LIN {X 0,Y 270.682,Z 565.079,A -85,B 0,C 180,E1 -18602.136,E2 -18602.136} C_VEL
LIN {X 0,Y 267.95,Z 577.412,A -85,B 0,C 180,E1 -18603.937,E2 -18603.937} C_VEL
LIN {X 0,Y 265.369,Z 587.551,A -85,B 0,C 180,E1 -18605.762,E2 -18605.762} C_VEL
LIN {X 0,Y 262.729,Z 597.619,A -85,B 0,C 180,E1 -18608.005,E2 -18608.005} C_VEL
LIN {X 0,Y 260.354,Z 605.98,A -85,B 0,C 180,E1 -18610.278,E2 -18610.278} C_VEL
LIN {X 0,Y 258.26,Z 613.967,A -85,B 0,C 180,E1 -18612.988,E2 -18612.988} C_VEL
LIN {X 0,Y 257.055,Z 618.72,A -85,B 0,C 180,E1 -18614.944,E2 -18614.944} C_VEL
LIN {X 0,Y 255.748,Z 623.456,A -85,B 0,C 180,E1 -18617.298,E2 -18617.298} C_VEL
LIN {X 0,Y 254.729,Z 628.359,A -85,B 0,C 180,E1 -18620.469,E2 -18620.469} C_VEL
LIN {X 0,Y 254.16,Z 631.774,A -85,B 0,C 180,E1 -18623.648,E2 -18623.648} C_VEL
LIN {X 0,Y 253.922,Z 633.804,A -85,B 0,C 180,E1 -18626.825,E2 -18626.825} C_VEL
LIN {X 0,Y 253.945,Z 634.498,A -85,B 0,C 180,E1 -18629.998,E2 -18629.998} C_VEL
LIN {X 0,Y 253.921,Z 633.866,A -85,B 0,C 180,E1 -18633.171,E2 -18633.171} C_VEL
LIN {X 0,Y 254.158,Z 631.893,A -85,B 0,C 180,E1 -18636.348,E2 -18636.348} C_VEL
LIN {X 0,Y 254.724,Z 628.531,A -85,B 0,C 180,E1 -18639.527,E2 -18639.527} C_VEL
LIN {X 0,Y 255.718,Z 623.68,A -85,B 0,C 180,E1 -18642.699,E2 -18642.699} C_VEL
LIN {X 0,Y 257.545,Z 617.197,A -85,B 0,C 180,E1 -18645.834,E2 -18645.834} C_VEL
LIN {X 0,Y 259.188,Z 610.543,A -85,B 0,C 180,E1 -18648.369,E2 -18648.369} C_VEL
LIN {X 0,Y 261.415,Z 602.415,A -85,B 0,C 180,E1 -18650.866,E2 -18650.866} C_VEL
LIN {X 0,Y 263.884,Z 593.336,A -85,B 0,C 180,E1 -18653.129,E2 -18653.129} C_VEL
LIN {X 0,Y 266.775,Z 582.336,A -85,B 0,C 180,E1 -18655.344,E2 -18655.344} C_VEL
LIN {X 0,Y 269.468,Z 571.253,A -85,B 0,C 180,E1 -18657.132,E2 -18657.132} C_VEL
LIN {X 0,Y 271.722,Z 560.272,A -85,B 0,C 180,E1 -18658.584,E2 -18658.584} C_VEL
LIN {X 0,Y 273.816,Z 548.655,A -85,B 0,C 180,E1 -18659.819,E2 -18659.819} C_VEL
LIN {X 0,Y 275.788,Z 536.139,A -85,B 0,C 180,E1 -18660.851,E2 -18660.851} C_VEL
LIN {X 0,Y 277.465,Z 522.233,A -85,B 0,C 180,E1 -18661.705,E2 -18661.705} C_VEL
LIN {X 0,Y 278.662,Z 508.127,A -85,B 0,C 180,E1 -18662.276,E2 -18662.276} C_VEL
LIN {X 0,Y 282.069,Z 423.35,A -85,B 0,C 180,E1 -18664.395,E2 -18664.395} C_VEL
LIN {X 0,Y 281.708,Z 421.592,A -85,B 0,C 180,E1 -18664.499,E2 -18664.499} C_VEL
LIN {X 0,Y 275.516,Z 406.79,A -85,B 0,C 180,E1 -18665.852,E2 -18665.852} C_VEL
LIN {X 0,Y 268.504,Z 392.298,A -85,B 0,C 180,E1 -18667.416,E2 -18667.416} C_VEL
LIN {X 0,Y 262.239,Z 380.582,A -85,B 0,C 180,E1 -18668.873,E2 -18668.873} C_VEL
LIN {X 0,Y 257.627,Z 372.309,A -85,B 0,C 180,E1 -18670.051,E2 -18670.051} C_VEL
LIN {X 0,Y 256.183,Z 367.432,A -85,B 0,C 180,E1 -18672.208,E2 -18672.208} C_VEL
LIN {X 0,Y 256.111,Z 367.17,A -85,B 0,C 180,E1 -18675.515,E2 -18675.515} C_VEL
LIN {X 0,Y 256.146,Z 367.192,A -85,B 0,C 180,E1 -18677.575,E2 -18677.575} C_VEL
LIN {X 0,Y 255.514,Z 367.285,A -85,B 0,C 180,E1 -18678.888,E2 -18678.888} C_VEL
LIN {X 0,Y 252.632,Z 367.623,A -85,B 0,C 180,E1 -18681.027,E2 -18681.027} C_VEL
LIN {X 0,Y 250.17,Z 367.909,A -85,B 0,C 180,E1 -18682.768,E2 -18682.768} C_VEL
LIN {X 0,Y 249.129,Z 368.043,A -85,B 0,C 180,E1 -18684.12,E2 -18684.12} C_VEL
LIN {X 0,Y 249.055,Z 368.06,A -85,B 0,C 180,E1 -18684.578,E2 -18684.578} C_VEL
LIN {X 0,Y 249.032,Z 368.067,A -85,B 0,C 180,E1 -18687.843,E2 -18687.843} C_VEL
LIN {X 0,Y 249.077,Z 368.015,A -85,B 0,C 180,E1 -18691.336,E2 -18691.336} C_VEL
LIN {X 0,Y 249.147,Z 368.069,A -85,B 0,C 180,E1 -18694.968,E2 -18694.968} C_VEL
LIN {X 0,Y 249.101,Z 368.069,A -85,B 0,C 180,E1 -18700.211,E2 -18700.211} C_VEL
LIN {X 0,Y 249.233,Z 368.043,A -85,B 0,C 180,E1 -18703.621,E2 -18703.621} C_VEL
LIN {X 0,Y 249.244,Z 368.052,A -85,B 0,C 180,E1 -18708.616,E2 -18708.616} C_VEL
LIN {X 0,Y 249.472,Z 368.017,A -85,B 0,C 180,E1 -18711.902,E2 -18711.902} C_VEL
LIN {X 0,Y 249.428,Z 368.015,A -85,B 0,C 180,E1 -18716.769,E2 -18716.769} C_VEL
LIN {X 0,Y 249.735,Z 368.002,A -85,B 0,C 180,E1 -18720,E2 -18720} C_VEL
LIN {X 0,Y 249.428,Z 368.015,A -85,B 0,C 180,E1 -18723.23,E2 -18723.23} C_VEL
LIN {X 0,Y 249.472,Z 368.018,A -85,B 0,C 180,E1 -18728.097,E2 -18728.097} C_VEL
LIN {X 0,Y 249.243,Z 368.05,A -85,B 0,C 180,E1 -18731.384,E2 -18731.384} C_VEL
LIN {X 0,Y 249.232,Z 368.041,A -85,B 0,C 180,E1 -18736.379,E2 -18736.379} C_VEL
LIN {X 0,Y 249.078,Z 368.062,A -85,B 0,C 180,E1 -18741.519,E2 -18741.519} C_VEL
LIN {X 0,Y 249.12,Z 368.062,A -85,B 0,C 180,E1 -18745.483,E2 -18745.483} C_VEL
LIN {X 0,Y 249.045,Z 368.017,A -85,B 0,C 180,E1 -18748.982,E2 -18748.982} C_VEL
LIN {X 0,Y 249.024,Z 368.074,A -85,B 0,C 180,E1 -18752.427,E2 -18752.427} C_VEL
LIN {X 0,Y 249.066,Z 368.042,A -85,B 0,C 180,E1 -18756.339,E2 -18756.339} C_VEL
LIN {X 0,Y 249.077,Z 368.064,A -85,B 0,C 180,E1 -18760.464,E2 -18760.464} C_VEL
LIN {X 0,Y 249.089,Z 368.062,A -85,B 0,C 180,E1 -18762.816,E2 -18762.816} C_VEL
LIN {X 0,Y 249.124,Z 368.184,A -85,B 0,C 180,E1 -18766.624,E2 -18766.624} C_VEL
LIN {X 0,Y 250.316,Z 372.193,A -85,B 0,C 180,E1 -18768.548,E2 -18768.548} C_VEL
LIN {X 0,Y 252.81,Z 376.584,A -85,B 0,C 180,E1 -18769.283,E2 -18769.283} C_VEL
LIN {X 0,Y 260.86,Z 390.951,A -85,B 0,C 180,E1 -18771.287,E2 -18771.287} C_VEL
LIN {X 0,Y 269.178,Z 407.825,A -85,B 0,C 180,E1 -18773.246,E2 -18773.246} C_VEL
LIN {X 0,Y 275.708,Z 423.186,A -85,B 0,C 180,E1 -18774.736,E2 -18774.736} C_VEL
LIN {X 0,Y 276.16,Z 424.395,A -85,B 0,C 180,E1 -18774.84,E2 -18774.84} C_VEL
LIN {X 0,Y 273.32,Z 494.281,A -85,B 0,C 180,E1 -18776.602,E2 -18776.602} C_VEL
LIN {X 0,Y 272.36,Z 512.78,A -85,B 0,C 180,E1 -18777.143,E2 -18777.143} C_VEL
LIN {X 0,Y 270.901,Z 526.969,A -85,B 0,C 180,E1 -18777.818,E2 -18777.818} C_VEL
LIN {X 0,Y 268.863,Z 541.315,A -85,B 0,C 180,E1 -18778.812,E2 -18778.812} C_VEL
LIN {X 0,Y 266.816,Z 553.585,A -85,B 0,C 180,E1 -18779.972,E2 -18779.972} C_VEL
LIN {X 0,Y 264.174,Z 566.61,A -85,B 0,C 180,E1 -18781.546,E2 -18781.546} C_VEL
LIN {X 0,Y 261.583,Z 577.852,A -85,B 0,C 180,E1 -18783.257,E2 -18783.257} C_VEL
LIN {X 0,Y 258.835,Z 587.92,A -85,B 0,C 180,E1 -18785.113,E2 -18785.113} C_VEL
LIN {X 0,Y 256.075,Z 597.926,A -85,B 0,C 180,E1 -18787.406,E2 -18787.406} C_VEL
LIN {X 0,Y 253.629,Z 606.235,A -85,B 0,C 180,E1 -18789.737,E2 -18789.737} C_VEL
LIN {X 0,Y 251.44,Z 614.176,A -85,B 0,C 180,E1 -18792.516,E2 -18792.516} C_VEL
LIN {X 0,Y 249.673,Z 620.565,A -85,B 0,C 180,E1 -18795.327,E2 -18795.327} C_VEL
LIN {X 0,Y 248.162,Z 626.231,A -85,B 0,C 180,E1 -18798.568,E2 -18798.568} C_VEL
LIN {X 0,Y 247.298,Z 630.341,A -85,B 0,C 180,E1 -18801.833,E2 -18801.833} C_VEL
LIN {X 0,Y 246.921,Z 633.019,A -85,B 0,C 180,E1 -18805.104,E2 -18805.104} C_VEL
LIN {X 0,Y 246.858,Z 634.339,A -85,B 0,C 180,E1 -18808.371,E2 -18808.371} C_VEL
LIN {X 0,Y 246.858,Z 634.329,A -85,B 0,C 180,E1 -18811.633,E2 -18811.633} C_VEL
LIN {X 0,Y 246.913,Z 632.946,A -85,B 0,C 180,E1 -18814.983,E2 -18814.983} C_VEL
LIN {X 0,Y 247.458,Z 633.053,A -85,B 0,C 180,E1 -18818.166,E2 -18818.166} C_VEL
LIN {X 0,Y 248.592,Z 632.021,A -85,B 0,C 180,E1 -18821.416,E2 -18821.416} C_VEL
LIN {X 0,Y 249.395,Z 630.903,A -85,B 0,C 180,E1 -18823.031,E2 -18823.031} C_VEL
LIN {X 0,Y 251.688,Z 627.42,A -85,B 0,C 180,E1 -18826.216,E2 -18826.216} C_VEL
LIN {X 0,Y 253.829,Z 623.708,A -85,B 0,C 180,E1 -18828.569,E2 -18828.569} C_VEL
LIN {X 0,Y 256.914,Z 618.089,A -85,B 0,C 180,E1 -18831.271,E2 -18831.271} C_VEL
LIN {X 0,Y 260.612,Z 610.935,A -85,B 0,C 180,E1 -18833.862,E2 -18833.862} C_VEL
LIN {X 0,Y 264.15,Z 603.407,A -85,B 0,C 180,E1 -18836.042,E2 -18836.042} C_VEL
LIN {X 0,Y 268.285,Z 594.335,A -85,B 0,C 180,E1 -18838.135,E2 -18838.135} C_VEL
LIN {X 0,Y 273.123,Z 582.307,A -85,B 0,C 180,E1 -18840.333,E2 -18840.333} C_VEL
LIN {X 0,Y 277.534,Z 569.741,A -85,B 0,C 180,E1 -18842.128,E2 -18842.128} C_VEL
LIN {X 0,Y 281.533,Z 556.94,A -85,B 0,C 180,E1 -18843.528,E2 -18843.528} C_VEL
LIN {X 0,Y 284.975,Z 543.739,A -85,B 0,C 180,E1 -18844.666,E2 -18844.666} C_VEL
LIN {X 0,Y 287.993,Z 529.205,A -85,B 0,C 180,E1 -18845.584,E2 -18845.584} C_VEL
LIN {X 0,Y 293.69,Z 498.987,A -85,B 0,C 180,E1 -18847.014,E2 -18847.014} C_VEL
LIN {X 0,Y 303.927,Z 448.446,A -85,B 0,C 180,E1 -18849.271,E2 -18849.271} C_VEL
LIN {X 0,Y 302.462,Z 446.463,A -85,B 0,C 180,E1 -18851.173,E2 -18851.173} C_VEL
LIN {X 0,Y 301.657,Z 446.072,A -85,B 0,C 180,E1 -18852.506,E2 -18852.506} C_VEL
LIN {X 0,Y 300.928,Z 446.396,A -85,B 0,C 180,E1 -18854.681,E2 -18854.681} C_VEL
LIN {X 0,Y 300.93,Z 448.238,A -85,B 0,C 180,E1 -18856.889,E2 -18856.889} C_VEL
LIN {X 0,Y 301.463,Z 451.187,A -85,B 0,C 180,E1 -18858.864,E2 -18858.864} C_VEL
LIN {X 0,Y 302.342,Z 455.625,A -85,B 0,C 180,E1 -18860.692,E2 -18860.692} C_VEL
LIN {X 0,Y 302.432,Z 456.877,A -85,B 0,C 180,E1 -18861,E2 -18861} C_VEL
LIN {X 0,Y 301.825,Z 467.626,A -85,B 0,C 180,E1 -18862.444,E2 -18862.444} C_VEL
LIN {X 0,Y 301.379,Z 474.057,A -85,B 0,C 180,E1 -18863.17,E2 -18863.17} C_VEL
LIN {X 0,Y 290.331,Z 534.975,A -85,B 0,C 180,E1 -18865.907,E2 -18865.907} C_VEL
LIN {X 0,Y 286.874,Z 549.388,A -85,B 0,C 180,E1 -18866.812,E2 -18866.812} C_VEL
LIN {X 0,Y 282.945,Z 562.72,A -85,B 0,C 180,E1 -18867.932,E2 -18867.932} C_VEL
LIN {X 0,Y 278.832,Z 574.736,A -85,B 0,C 180,E1 -18869.274,E2 -18869.274} C_VEL
LIN {X 0,Y 275.145,Z 584.325,A -85,B 0,C 180,E1 -18870.604,E2 -18870.604} C_VEL
LIN {X 0,Y 270.491,Z 595.122,A -85,B 0,C 180,E1 -18872.467,E2 -18872.467} C_VEL
LIN {X 0,Y 265.961,Z 604.624,A -85,B 0,C 180,E1 -18874.57,E2 -18874.57} C_VEL
LIN {X 0,Y 261.96,Z 612.26,A -85,B 0,C 180,E1 -18876.689,E2 -18876.689} C_VEL
LIN {X 0,Y 257.888,Z 619.427,A -85,B 0,C 180,E1 -18879.251,E2 -18879.251} C_VEL
LIN {X 0,Y 255.004,Z 624.276,A -85,B 0,C 180,E1 -18881.522,E2 -18881.522} C_VEL
LIN {X 0,Y 252.691,Z 628.054,A -85,B 0,C 180,E1 -18883.852,E2 -18883.852} C_VEL
LIN {X 0,Y 250.104,Z 631.618,A -85,B 0,C 180,E1 -18887.009,E2 -18887.009} C_VEL
LIN {X 0,Y 249.081,Z 632.779,A -85,B 0,C 180,E1 -18888.609,E2 -18888.609} C_VEL
LIN {X 0,Y 247.692,Z 633.851,A -85,B 0,C 180,E1 -18891.844,E2 -18891.844} C_VEL
LIN {X 0,Y 247.059,Z 633.485,A -85,B 0,C 180,E1 -18894.659,E2 -18894.659} C_VEL
LIN {X 0,Y 246.938,Z 632.417,A -85,B 0,C 180,E1 -18896.737,E2 -18896.737} C_VEL
LIN {X 0,Y 246.954,Z 631.103,A -85,B 0,C 180,E1 -18898.369,E2 -18898.369} C_VEL
LIN {X 0,Y 246.922,Z 628.265,A -85,B 0,C 180,E1 -18900.816,E2 -18900.816} C_VEL
LIN {X 0,Y 247.116,Z 624.344,A -85,B 0,C 180,E1 -18903.261,E2 -18903.261} C_VEL
LIN {X 0,Y 247.256,Z 618.937,A -85,B 0,C 180,E1 -18905.808,E2 -18905.808} C_VEL
LIN {X 0,Y 247.653,Z 611.315,A -85,B 0,C 180,E1 -18908.568,E2 -18908.568} C_VEL
LIN {X 0,Y 248.166,Z 602.752,A -85,B 0,C 180,E1 -18911.021,E2 -18911.021} C_VEL
LIN {X 0,Y 249.031,Z 592.004,A -85,B 0,C 180,E1 -18913.464,E2 -18913.464} C_VEL
LIN {X 0,Y 249.973,Z 580.808,A -85,B 0,C 180,E1 -18915.491,E2 -18915.491} C_VEL
LIN {X 0,Y 250.907,Z 569.831,A -85,B 0,C 180,E1 -18917.104,E2 -18917.104} C_VEL
LIN {X 0,Y 251.878,Z 557.647,A -85,B 0,C 180,E1 -18918.524,E2 -18918.524} C_VEL
LIN {X 0,Y 252.724,Z 544.556,A -85,B 0,C 180,E1 -18919.706,E2 -18919.706} C_VEL
LIN {X 0,Y 253.625,Z 530.023,A -85,B 0,C 180,E1 -18920.637,E2 -18920.637} C_VEL
LIN {X 0,Y 256.52,Z 454.942,A -85,B 0,C 180,E1 -18924.024,E2 -18924.024} C_VEL
LIN {X 0,Y 254.21,Z 430.351,A -85,B 0,C 180,E1 -18925.232,E2 -18925.232} C_VEL
LIN {X 0,Y 253.707,Z 419.989,A -85,B 0,C 180,E1 -18925.763,E2 -18925.763} C_VEL
LIN {X 0,Y 255.862,Z 399.784,A -85,B 0,C 180,E1 -18930.086,E2 -18930.086} C_VEL
LIN {X 0,Y 255.22,Z 395.695,A -85,B 0,C 180,E1 -18931.029,E2 -18931.029} C_VEL
LIN {X 0,Y 251.804,Z 380.115,A -85,B 0,C 180,E1 -18934.747,E2 -18934.747} C_VEL
LIN {X 0,Y 249.15,Z 368.273,A -85,B 0,C 180,E1 -18937.727,E2 -18937.727} C_VEL
LIN {X 0,Y 249.007,Z 368.076,A -85,B 0,C 180,E1 -18942.789,E2 -18942.789} C_VEL
LIN {X 0,Y 249.022,Z 368.134,A -85,B 0,C 180,E1 -18946.639,E2 -18946.639} C_VEL
LIN {X 0,Y 249.878,Z 371.102,A -85,B 0,C 180,E1 -18948.201,E2 -18948.201} C_VEL
LIN {X 0,Y 250.419,Z 372.631,A -85,B 0,C 180,E1 -18948.736,E2 -18948.736} C_VEL
LIN {X 0,Y 252.743,Z 376.544,A -85,B 0,C 180,E1 -18949.37,E2 -18949.37} C_VEL
LIN {X 0,Y 261.085,Z 391.423,A -85,B 0,C 180,E1 -18951.439,E2 -18951.439} C_VEL
LIN {X 0,Y 268.827,Z 407.158,A -85,B 0,C 180,E1 -18953.26,E2 -18953.26} C_VEL
LIN {X 0,Y 275.079,Z 421.704,A -85,B 0,C 180,E1 -18954.684,E2 -18954.684} C_VEL
LIN {X 0,Y 275.984,Z 424.12,A -85,B 0,C 180,E1 -18954.892,E2 -18954.892} C_VEL
LIN {X 0,Y 273.318,Z 492.571,A -85,B 0,C 180,E1 -18956.635,E2 -18956.635} C_VEL
LIN {X 0,Y 272.335,Z 511.911,A -85,B 0,C 180,E1 -18957.183,E2 -18957.183} C_VEL
LIN {X 0,Y 270.868,Z 526.495,A -85,B 0,C 180,E1 -18957.864,E2 -18957.864} C_VEL
LIN {X 0,Y 269.113,Z 539.27,A -85,B 0,C 180,E1 -18958.73,E2 -18958.73} C_VEL
LIN {X 0,Y 266.839,Z 552.859,A -85,B 0,C 180,E1 -18959.97,E2 -18959.97} C_VEL
LIN {X 0,Y 264.394,Z 565.083,A -85,B 0,C 180,E1 -18961.413,E2 -18961.413} C_VEL
LIN {X 0,Y 261.581,Z 577.415,A -85,B 0,C 180,E1 -18963.253,E2 -18963.253} C_VEL
LIN {X 0,Y 258.897,Z 587.554,A -85,B 0,C 180,E1 -18965.115,E2 -18965.115} C_VEL
LIN {X 0,Y 256.118,Z 597.622,A -85,B 0,C 180,E1 -18967.406,E2 -18967.406} C_VEL
LIN {X 0,Y 253.664,Z 605.982,A -85,B 0,C 180,E1 -18969.735,E2 -18969.735} C_VEL
LIN {X 0,Y 251.447,Z 613.969,A -85,B 0,C 180,E1 -18972.513,E2 -18972.513} C_VEL
LIN {X 0,Y 249.685,Z 620.402,A -85,B 0,C 180,E1 -18975.324,E2 -18975.324} C_VEL
LIN {X 0,Y 248.175,Z 626.103,A -85,B 0,C 180,E1 -18978.564,E2 -18978.564} C_VEL
LIN {X 0,Y 247.301,Z 630.245,A -85,B 0,C 180,E1 -18981.829,E2 -18981.829} C_VEL
LIN {X 0,Y 246.923,Z 632.958,A -85,B 0,C 180,E1 -18985.1,E2 -18985.1} C_VEL
LIN {X 0,Y 246.859,Z 634.317,A -85,B 0,C 180,E1 -18988.367,E2 -18988.367} C_VEL
LIN {X 0,Y 246.858,Z 634.348,A -85,B 0,C 180,E1 -18991.629,E2 -18991.629} C_VEL
LIN {X 0,Y 246.913,Z 632.993,A -85,B 0,C 180,E1 -18994.979,E2 -18994.979} C_VEL
LIN {X 0,Y 247.298,Z 630.39,A -85,B 0,C 180,E1 -18998.167,E2 -18998.167} C_VEL
LIN {X 0,Y 248.158,Z 626.299,A -85,B 0,C 180,E1 -19001.432,E2 -19001.432} C_VEL
LIN {X 0,Y 249.656,Z 620.652,A -85,B 0,C 180,E1 -19004.674,E2 -19004.674} C_VEL
LIN {X 0,Y 251.429,Z 614.284,A -85,B 0,C 180,E1 -19007.485,E2 -19007.485} C_VEL
LIN {X 0,Y 253.633,Z 606.366,A -85,B 0,C 180,E1 -19010.263,E2 -19010.263} C_VEL
LIN {X 0,Y 256.009,Z 598.083,A -85,B 0,C 180,E1 -19012.6,E2 -19012.6} C_VEL
LIN {X 0,Y 258.781,Z 588.107,A -85,B 0,C 180,E1 -19014.892,E2 -19014.892} C_VEL
LIN {X 0,Y 261.743,Z 577,A -85,B 0,C 180,E1 -19016.941,E2 -19016.941} C_VEL
LIN {X 0,Y 264.519,Z 564.813,A -85,B 0,C 180,E1 -19018.744,E2 -19018.744} C_VEL
LIN {X 0,Y 267.037,Z 552.183,A -85,B 0,C 180,E1 -19020.219,E2 -19020.219} C_VEL
LIN {X 0,Y 269.337,Z 538.391,A -85,B 0,C 180,E1 -19021.455,E2 -19021.455} C_VEL
LIN {X 0,Y 271.191,Z 524.547,A -85,B 0,C 180,E1 -19022.363,E2 -19022.363} C_VEL
LIN {X 0,Y 272.491,Z 510.628,A -85,B 0,C 180,E1 -19022.989,E2 -19022.989} C_VEL
LIN {X 0,Y 274.083,Z 477.516,A -85,B 0,C 180,E1 -19023.854,E2 -19023.854} C_VEL
LIN {X 0,Y 276.114,Z 424.266,A -85,B 0,C 180,E1 -19025.216,E2 -19025.216} C_VEL
LIN {X 0,Y 270.167,Z 410.023,A -85,B 0,C 180,E1 -19026.571,E2 -19026.571} C_VEL
LIN {X 0,Y 263.041,Z 395.254,A -85,B 0,C 180,E1 -19028.231,E2 -19028.231} C_VEL
LIN {X 0,Y 257.206,Z 384.361,A -85,B 0,C 180,E1 -19029.647,E2 -19029.647} C_VEL
LIN {X 0,Y 251.959,Z 375.375,A -85,B 0,C 180,E1 -19030.974,E2 -19030.974} C_VEL
LIN {X 0,Y 250.283,Z 372.109,A -85,B 0,C 180,E1 -19031.516,E2 -19031.516} C_VEL
LIN {X 0,Y 249.125,Z 368.232,A -85,B 0,C 180,E1 -19033.376,E2 -19033.376} C_VEL
LIN {X 0,Y 249.08,Z 368.065,A -85,B 0,C 180,E1 -19037.547,E2 -19037.547} C_VEL
LIN {X 0,Y 249.045,Z 368.037,A -85,B 0,C 180,E1 -19041.623,E2 -19041.623} C_VEL
LIN {X 0,Y 249.055,Z 368.06,A -85,B 0,C 180,E1 -19044.578,E2 -19044.578} C_VEL
LIN {X 0,Y 248.405,Z 368.169,A -85,B 0,C 180,E1 -19045.927,E2 -19045.927} C_VEL
LIN {X 0,Y 245.531,Z 368.495,A -85,B 0,C 180,E1 -19048.124,E2 -19048.124} C_VEL
LIN {X 0,Y 243.084,Z 368.77,A -85,B 0,C 180,E1 -19049.914,E2 -19049.914} C_VEL
LIN {X 0,Y 242.05,Z 368.889,A -85,B 0,C 180,E1 -19051.304,E2 -19051.304} C_VEL
LIN {X 0,Y 241.974,Z 368.9,A -85,B 0,C 180,E1 -19051.775,E2 -19051.775} C_VEL
LIN {X 0,Y 242.059,Z 368.933,A -85,B 0,C 180,E1 -19054.182,E2 -19054.182} C_VEL
LIN {X 0,Y 242.044,Z 368.94,A -85,B 0,C 180,E1 -19058.296,E2 -19058.296} C_VEL
LIN {X 0,Y 242.154,Z 368.928,A -85,B 0,C 180,E1 -19063.277,E2 -19063.277} C_VEL
LIN {X 0,Y 242.177,Z 368.937,A -85,B 0,C 180,E1 -19068.279,E2 -19068.279} C_VEL
LIN {X 0,Y 242.418,Z 368.892,A -85,B 0,C 180,E1 -19071.665,E2 -19071.665} C_VEL
LIN {X 0,Y 242.253,Z 368.922,A -85,B 0,C 180,E1 -19075.007,E2 -19075.007} C_VEL
LIN {X 0,Y 242.628,Z 368.873,A -85,B 0,C 180,E1 -19078.34,E2 -19078.34} C_VEL
LIN {X 0,Y 242.628,Z 368.874,A -85,B 0,C 180,E1 -19081.66,E2 -19081.66} C_VEL
LIN {X 0,Y 242.424,Z 368.912,A -85,B 0,C 180,E1 -19086.659,E2 -19086.659} C_VEL
LIN {X 0,Y 242.304,Z 368.901,A -85,B 0,C 180,E1 -19090.022,E2 -19090.022} C_VEL
LIN {X 0,Y 242.157,Z 368.919,A -85,B 0,C 180,E1 -19095.141,E2 -19095.141} C_VEL
LIN {X 0,Y 242.064,Z 368.955,A -85,B 0,C 180,E1 -19098.625,E2 -19098.625} C_VEL
LIN {X 0,Y 242.004,Z 368.946,A -85,B 0,C 180,E1 -19102.181,E2 -19102.181} C_VEL
LIN {X 0,Y 242.057,Z 368.932,A -85,B 0,C 180,E1 -19105.839,E2 -19105.839} C_VEL
LIN {X 0,Y 241.966,Z 368.899,A -85,B 0,C 180,E1 -19109.589,E2 -19109.589} C_VEL
LIN {X 0,Y 241.981,Z 368.969,A -85,B 0,C 180,E1 -19113.492,E2 -19113.492} C_VEL
LIN {X 0,Y 242.004,Z 368.911,A -85,B 0,C 180,E1 -19117.579,E2 -19117.579} C_VEL
LIN {X 0,Y 242.031,Z 368.96,A -85,B 0,C 180,E1 -19121.902,E2 -19121.902} C_VEL
LIN {X 0,Y 242.037,Z 369.119,A -85,B 0,C 180,E1 -19125.462,E2 -19125.462} C_VEL
LIN {X 0,Y 242.96,Z 372.191,A -85,B 0,C 180,E1 -19126.992,E2 -19126.992} C_VEL
LIN {X 0,Y 245.645,Z 376.648,A -85,B 0,C 180,E1 -19127.83,E2 -19127.83} C_VEL
LIN {X 0,Y 253.86,Z 390.901,A -85,B 0,C 180,E1 -19130.007,E2 -19130.007} C_VEL
LIN {X 0,Y 261.86,Z 406.738,A -85,B 0,C 180,E1 -19132.003,E2 -19132.003} C_VEL
LIN {X 0,Y 268.962,Z 422.871,A -85,B 0,C 180,E1 -19133.702,E2 -19133.702} C_VEL
LIN {X 0,Y 270.265,Z 426.248,A -85,B 0,C 180,E1 -19134.014,E2 -19134.014} C_VEL
LIN {X 0,Y 267.477,Z 493.79,A -85,B 0,C 180,E1 -19135.757,E2 -19135.757} C_VEL
LIN {X 0,Y 266.519,Z 511.884,A -85,B 0,C 180,E1 -19136.282,E2 -19136.282} C_VEL
LIN {X 0,Y 265.053,Z 526.216,A -85,B 0,C 180,E1 -19136.963,E2 -19136.963} C_VEL
LIN {X 0,Y 263.014,Z 540.192,A -85,B 0,C 180,E1 -19137.924,E2 -19137.924} C_VEL
LIN {X 0,Y 260.685,Z 553.591,A -85,B 0,C 180,E1 -19139.19,E2 -19139.19} C_VEL
LIN {X 0,Y 258.141,Z 565.669,A -85,B 0,C 180,E1 -19140.658,E2 -19140.658} C_VEL
LIN {X 0,Y 255.251,Z 577.855,A -85,B 0,C 180,E1 -19142.539,E2 -19142.539} C_VEL
LIN {X 0,Y 252.401,Z 587.923,A -85,B 0,C 180,E1 -19144.434,E2 -19144.434} C_VEL
LIN {X 0,Y 249.515,Z 597.928,A -85,B 0,C 180,E1 -19146.778,E2 -19146.778} C_VEL
LIN {X 0,Y 246.935,Z 606.237,A -85,B 0,C 180,E1 -19149.162,E2 -19149.162} C_VEL
LIN {X 0,Y 244.644,Z 614.178,A -85,B 0,C 180,E1 -19152.014,E2 -19152.014} C_VEL
LIN {X 0,Y 242.771,Z 620.567,A -85,B 0,C 180,E1 -19154.9,E2 -19154.9} C_VEL
LIN {X 0,Y 241.485,Z 624.99,A -85,B 0,C 180,E1 -19157.395,E2 -19157.395} C_VEL
LIN {X 0,Y 240.664,Z 628.473,A -85,B 0,C 180,E1 -19159.911,E2 -19159.911} C_VEL
LIN {X 0,Y 239.995,Z 631.853,A -85,B 0,C 180,E1 -19163.275,E2 -19163.275} C_VEL
LIN {X 0,Y 239.742,Z 633.846,A -85,B 0,C 180,E1 -19166.641,E2 -19166.641} C_VEL
LIN {X 0,Y 239.772,Z 634.339,A -85,B 0,C 180,E1 -19168.322,E2 -19168.322} C_VEL
LIN {X 0,Y 239.771,Z 634.329,A -85,B 0,C 180,E1 -19171.682,E2 -19171.682} C_VEL
LIN {X 0,Y 239.841,Z 632.992,A -85,B 0,C 180,E1 -19175.045,E2 -19175.045} C_VEL
LIN {X 0,Y 239.91,Z 632.611,A -85,B 0,C 180,E1 -19175.887,E2 -19175.887} C_VEL
LIN {X 0,Y 240.422,Z 633.111,A -85,B 0,C 180,E1 -19178.407,E2 -19178.407} C_VEL
LIN {X 0,Y 240.919,Z 632.934,A -85,B 0,C 180,E1 -19180.082,E2 -19180.082} C_VEL
LIN {X 0,Y 242.497,Z 631.399,A -85,B 0,C 180,E1 -19183.408,E2 -19183.408} C_VEL
LIN {X 0,Y 243.619,Z 630.058,A -85,B 0,C 180,E1 -19185.05,E2 -19185.05} C_VEL
LIN {X 0,Y 246.37,Z 626.136,A -85,B 0,C 180,E1 -19188.29,E2 -19188.29} C_VEL
LIN {X 0,Y 248.976,Z 622.079,A -85,B 0,C 180,E1 -19190.663,E2 -19190.663} C_VEL
LIN {X 0,Y 252.556,Z 616.144,A -85,B 0,C 180,E1 -19193.32,E2 -19193.32} C_VEL
LIN {X 0,Y 256.856,Z 608.447,A -85,B 0,C 180,E1 -19195.965,E2 -19195.965} C_VEL
LIN {X 0,Y 260.951,Z 600.44,A -85,B 0,C 180,E1 -19198.122,E2 -19198.122} C_VEL
LIN {X 0,Y 265.54,Z 590.865,A -85,B 0,C 180,E1 -19200.192,E2 -19200.192} C_VEL
LIN {X 0,Y 270.52,Z 579.19,A -85,B 0,C 180,E1 -19202.182,E2 -19202.182} C_VEL
LIN {X 0,Y 274.443,Z 568.729,A -85,B 0,C 180,E1 -19203.628,E2 -19203.628} C_VEL
LIN {X 0,Y 278.766,Z 555.819,A -85,B 0,C 180,E1 -19205,E2 -19205} C_VEL
LIN {X 0,Y 282.459,Z 542.499,A -85,B 0,C 180,E1 -19206.115,E2 -19206.115} C_VEL
LIN {X 0,Y 285.605,Z 528.442,A -85,B 0,C 180,E1 -19206.968,E2 -19206.968} C_VEL
LIN {X 0,Y 291.288,Z 500.27,A -85,B 0,C 180,E1 -19208.301,E2 -19208.301} C_VEL
LIN {X 0,Y 301.184,Z 454.187,A -85,B 0,C 180,E1 -19210.349,E2 -19210.349} C_VEL
LIN {X 0,Y 300.424,Z 453.169,A -85,B 0,C 180,E1 -19211.531,E2 -19211.531} C_VEL
LIN {X 0,Y 299.275,Z 453.094,A -85,B 0,C 180,E1 -19214.135,E2 -19214.135} C_VEL
LIN {X 0,Y 299.063,Z 454.758,A -85,B 0,C 180,E1 -19216.486,E2 -19216.486} C_VEL
LIN {X 0,Y 299.43,Z 457.574,A -85,B 0,C 180,E1 -19218.415,E2 -19218.415} C_VEL
LIN {X 0,Y 299.998,Z 461.533,A -85,B 0,C 180,E1 -19220.077,E2 -19220.077} C_VEL
LIN {X 0,Y 299.102,Z 471.743,A -85,B 0,C 180,E1 -19221.45,E2 -19221.45} C_VEL
LIN {X 0,Y 298.754,Z 475.787,A -85,B 0,C 180,E1 -19221.938,E2 -19221.938} C_VEL
LIN {X 0,Y 287.104,Z 535.821,A -85,B 0,C 180,E1 -19224.668,E2 -19224.668} C_VEL
LIN {X 0,Y 283.76,Z 548.923,A -85,B 0,C 180,E1 -19225.49,E2 -19225.49} C_VEL
LIN {X 0,Y 280.007,Z 561.066,A -85,B 0,C 180,E1 -19226.483,E2 -19226.483} C_VEL
LIN {X 0,Y 275.492,Z 573.524,A -85,B 0,C 180,E1 -19227.817,E2 -19227.817} C_VEL
LIN {X 0,Y 270.987,Z 584.456,A -85,B 0,C 180,E1 -19229.323,E2 -19229.323} C_VEL
LIN {X 0,Y 266.081,Z 595.118,A -85,B 0,C 180,E1 -19231.182,E2 -19231.182} C_VEL
LIN {X 0,Y 261.349,Z 604.297,A -85,B 0,C 180,E1 -19233.229,E2 -19233.229} C_VEL
LIN {X 0,Y 256.996,Z 611.964,A -85,B 0,C 180,E1 -19235.352,E2 -19235.352} C_VEL
LIN {X 0,Y 252.57,Z 619.141,A -85,B 0,C 180,E1 -19237.936,E2 -19237.936} C_VEL
LIN {X 0,Y 249.25,Z 624.037,A -85,B 0,C 180,E1 -19240.223,E2 -19240.223} C_VEL
LIN {X 0,Y 245.918,Z 628.902,A -85,B 0,C 180,E1 -19243.394,E2 -19243.394} C_VEL
LIN {X 0,Y 244.458,Z 630.712,A -85,B 0,C 180,E1 -19245.005,E2 -19245.005} C_VEL
LIN {X 0,Y 242.12,Z 633.077,A -85,B 0,C 180,E1 -19248.277,E2 -19248.277} C_VEL
LIN {X 0,Y 241.291,Z 633.679,A -85,B 0,C 180,E1 -19249.935,E2 -19249.935} C_VEL
LIN {X 0,Y 240.668,Z 633.877,A -85,B 0,C 180,E1 -19251.604,E2 -19251.604} C_VEL
LIN {X 0,Y 239.955,Z 633.016,A -85,B 0,C 180,E1 -19254.959,E2 -19254.959} C_VEL
LIN {X 0,Y 239.864,Z 631.997,A -85,B 0,C 180,E1 -19256.641,E2 -19256.641} C_VEL
LIN {X 0,Y 239.887,Z 630.545,A -85,B 0,C 180,E1 -19258.321,E2 -19258.321} C_VEL
LIN {X 0,Y 239.86,Z 627.491,A -85,B 0,C 180,E1 -19260.84,E2 -19260.84} C_VEL
LIN {X 0,Y 240.064,Z 623.319,A -85,B 0,C 180,E1 -19263.357,E2 -19263.357} C_VEL
LIN {X 0,Y 240.238,Z 616.815,A -85,B 0,C 180,E1 -19266.298,E2 -19266.298} C_VEL
LIN {X 0,Y 240.622,Z 609.675,A -85,B 0,C 180,E1 -19268.821,E2 -19268.821} C_VEL
LIN {X 0,Y 241.209,Z 600.678,A -85,B 0,C 180,E1 -19271.343,E2 -19271.343} C_VEL
LIN {X 0,Y 242.023,Z 590.478,A -85,B 0,C 180,E1 -19273.647,E2 -19273.647} C_VEL
LIN {X 0,Y 243.019,Z 579.023,A -85,B 0,C 180,E1 -19275.731,E2 -19275.731} C_VEL
LIN {X 0,Y 243.987,Z 567.651,A -85,B 0,C 180,E1 -19277.379,E2 -19277.379} C_VEL
LIN {X 0,Y 244.943,Z 555.096,A -85,B 0,C 180,E1 -19278.827,E2 -19278.827} C_VEL
LIN {X 0,Y 245.886,Z 540.868,A -85,B 0,C 180,E1 -19280.059,E2 -19280.059} C_VEL
LIN {X 0,Y 246.633,Z 526.683,A -85,B 0,C 180,E1 -19280.922,E2 -19280.922} C_VEL
LIN {X 0,Y 249.531,Z 455.682,A -85,B 0,C 180,E1 -19284.237,E2 -19284.237} C_VEL
LIN {X 0,Y 247.272,Z 431.277,A -85,B 0,C 180,E1 -19285.489,E2 -19285.489} C_VEL
LIN {X 0,Y 246.724,Z 419.879,A -85,B 0,C 180,E1 -19286.088,E2 -19286.088} C_VEL
LIN {X 0,Y 248.883,Z 400.533,A -85,B 0,C 180,E1 -19290.316,E2 -19290.316} C_VEL
LIN {X 0,Y 246.277,Z 387.884,A -85,B 0,C 180,E1 -19293.359,E2 -19293.359} C_VEL
LIN {X 0,Y 242.339,Z 370.216,A -85,B 0,C 180,E1 -19297.761,E2 -19297.761} C_VEL
LIN {X 0,Y 242.085,Z 369.085,A -85,B 0,C 180,E1 -19298.157,E2 -19298.157} C_VEL
LIN {X 0,Y 241.931,Z 368.946,A -85,B 0,C 180,E1 -19303.425,E2 -19303.425} C_VEL
LIN {X 0,Y 241.97,Z 368.98,A -85,B 0,C 180,E1 -19305.429,E2 -19305.429} C_VEL
LIN {X 0,Y 242.673,Z 371.514,A -85,B 0,C 180,E1 -19306.817,E2 -19306.817} C_VEL
LIN {X 0,Y 243.005,Z 372.492,A -85,B 0,C 180,E1 -19307.165,E2 -19307.165} C_VEL
LIN {X 0,Y 249.627,Z 383.55,A -85,B 0,C 180,E1 -19309.015,E2 -19309.015} C_VEL
LIN {X 0,Y 256.388,Z 395.727,A -85,B 0,C 180,E1 -19310.749,E2 -19310.749} C_VEL
LIN {X 0,Y 264.091,Z 411.671,A -85,B 0,C 180,E1 -19312.639,E2 -19312.639} C_VEL
LIN {X 0,Y 268.95,Z 423.104,A -85,B 0,C 180,E1 -19313.798,E2 -19313.798} C_VEL
LIN {X 0,Y 270.206,Z 426.248,A -85,B 0,C 180,E1 -19314.094,E2 -19314.094} C_VEL
LIN {X 0,Y 266.701,Z 508.068,A -85,B 0,C 180,E1 -19316.219,E2 -19316.219} C_VEL
LIN {X 0,Y 265.368,Z 522.69,A -85,B 0,C 180,E1 -19316.833,E2 -19316.833} C_VEL
LIN {X 0,Y 263.408,Z 537.02,A -85,B 0,C 180,E1 -19317.748,E2 -19317.748} C_VEL
LIN {X 0,Y 261.362,Z 549.336,A -85,B 0,C 180,E1 -19318.825,E2 -19318.825} C_VEL
LIN {X 0,Y 258.694,Z 562.525,A -85,B 0,C 180,E1 -19320.321,E2 -19320.321} C_VEL
LIN {X 0,Y 255.817,Z 575.121,A -85,B 0,C 180,E1 -19322.156,E2 -19322.156} C_VEL
LIN {X 0,Y 252.99,Z 585.637,A -85,B 0,C 180,E1 -19324.052,E2 -19324.052} C_VEL
LIN {X 0,Y 250.001,Z 596.084,A -85,B 0,C 180,E1 -19326.383,E2 -19326.383} C_VEL
LIN {X 0,Y 247.403,Z 604.701,A -85,B 0,C 180,E1 -19328.763,E2 -19328.763} C_VEL
LIN {X 0,Y 244.945,Z 612.961,A -85,B 0,C 180,E1 -19331.6,E2 -19331.6} C_VEL
LIN {X 0,Y 243.318,Z 618.723,A -85,B 0,C 180,E1 -19334.072,E2 -19334.072} C_VEL
LIN {X 0,Y 241.835,Z 623.459,A -85,B 0,C 180,E1 -19336.554,E2 -19336.554} C_VEL
LIN {X 0,Y 240.67,Z 628.361,A -85,B 0,C 180,E1 -19339.907,E2 -19339.907} C_VEL
LIN {X 0,Y 239.997,Z 631.775,A -85,B 0,C 180,E1 -19343.271,E2 -19343.271} C_VEL
LIN {X 0,Y 239.741,Z 633.804,A -85,B 0,C 180,E1 -19346.637,E2 -19346.637} C_VEL
LIN {X 0,Y 239.773,Z 634.318,A -85,B 0,C 180,E1 -19348.318,E2 -19348.318} C_VEL
LIN {X 0,Y 239.772,Z 634.348,A -85,B 0,C 180,E1 -19351.678,E2 -19351.678} C_VEL
LIN {X 0,Y 239.841,Z 633.049,A -85,B 0,C 180,E1 -19355.041,E2 -19355.041} C_VEL
LIN {X 0,Y 240.243,Z 630.389,A -85,B 0,C 180,E1 -19358.409,E2 -19358.409} C_VEL
LIN {X 0,Y 241.176,Z 626.298,A -85,B 0,C 180,E1 -19361.768,E2 -19361.768} C_VEL
LIN {X 0,Y 242.752,Z 620.651,A -85,B 0,C 180,E1 -19365.101,E2 -19365.101} C_VEL
LIN {X 0,Y 244.642,Z 614.282,A -85,B 0,C 180,E1 -19367.986,E2 -19367.986} C_VEL
LIN {X 0,Y 246.932,Z 606.364,A -85,B 0,C 180,E1 -19370.838,E2 -19370.838} C_VEL
LIN {X 0,Y 249.451,Z 598.081,A -85,B 0,C 180,E1 -19373.228,E2 -19373.228} C_VEL
LIN {X 0,Y 252.336,Z 588.104,A -85,B 0,C 180,E1 -19375.573,E2 -19375.573} C_VEL
LIN {X 0,Y 255.411,Z 576.996,A -85,B 0,C 180,E1 -19377.665,E2 -19377.665} C_VEL
LIN {X 0,Y 258.327,Z 564.681,A -85,B 0,C 180,E1 -19379.519,E2 -19379.519} C_VEL
LIN {X 0,Y 260.919,Z 552.177,A -85,B 0,C 180,E1 -19381.004,E2 -19381.004} C_VEL
LIN {X 0,Y 263.315,Z 538.383,A -85,B 0,C 180,E1 -19382.261,E2 -19382.261} C_VEL
LIN {X 0,Y 265.218,Z 524.536,A -85,B 0,C 180,E1 -19383.184,E2 -19383.184} C_VEL
LIN {X 0,Y 266.557,Z 510.786,A -85,B 0,C 180,E1 -19383.812,E2 -19383.812} C_VEL
LIN {X 0,Y 268.153,Z 479.267,A -85,B 0,C 180,E1 -19384.652,E2 -19384.652} C_VEL
LIN {X 0,Y 270.249,Z 426.161,A -85,B 0,C 180,E1 -19386.037,E2 -19386.037} C_VEL
LIN {X 0,Y 263.648,Z 410.628,A -85,B 0,C 180,E1 -19387.608,E2 -19387.608} C_VEL
LIN {X 0,Y 255.341,Z 393.597,A -85,B 0,C 180,E1 -19389.663,E2 -19389.663} C_VEL
LIN {X 0,Y 247.739,Z 380.28,A -85,B 0,C 180,E1 -19391.64,E2 -19391.64} C_VEL
LIN {X 0,Y 244.865,Z 375.643,A -85,B 0,C 180,E1 -19392.42,E2 -19392.42} C_VEL
LIN {X 0,Y 242.896,Z 372.031,A -85,B 0,C 180,E1 -19393.102,E2 -19393.102} C_VEL
LIN {X 0,Y 242.05,Z 369.051,A -85,B 0,C 180,E1 -19394.641,E2 -19394.641} C_VEL
LIN {X 0,Y 242.006,Z 368.957,A -85,B 0,C 180,E1 -19399.026,E2 -19399.026} C_VEL
LIN {X 0,Y 242.005,Z 368.911,A -85,B 0,C 180,E1 -19402.421,E2 -19402.421} C_VEL
LIN {X 0,Y 241.984,Z 368.969,A -85,B 0,C 180,E1 -19406.508,E2 -19406.508} C_VEL
LIN {X 0,Y 242.005,Z 368.895,A -85,B 0,C 180,E1 -19410.596,E2 -19410.596} C_VEL
LIN {X 0,Y 241.974,Z 368.9,A -85,B 0,C 180,E1 -19411.775,E2 -19411.775} C_VEL
LIN {X 0,Y 241.346,Z 369.001,A -85,B 0,C 180,E1 -19413.164,E2 -19413.164} C_VEL
LIN {X 0,Y 238.559,Z 369.392,A -85,B 0,C 180,E1 -19415.43,E2 -19415.43} C_VEL
LIN {X 0,Y 235.335,Z 369.777,A -85,B 0,C 180,E1 -19418.224,E2 -19418.224} C_VEL
LIN {X 0,Y 234.989,Z 369.818,A -85,B 0,C 180,E1 -19419.192,E2 -19419.192} C_VEL
LIN {X 0,Y 235.087,Z 369.81,A -85,B 0,C 180,E1 -19423.059,E2 -19423.059} C_VEL
LIN {X 0,Y 235.138,Z 369.816,A -85,B 0,C 180,E1 -19427.923,E2 -19427.923} C_VEL
LIN {X 0,Y 235.367,Z 369.768,A -85,B 0,C 180,E1 -19431.414,E2 -19431.414} C_VEL
LIN {X 0,Y 235.395,Z 369.784,A -85,B 0,C 180,E1 -19433.141,E2 -19433.141} C_VEL
LIN {X 0,Y 235.588,Z 369.749,A -85,B 0,C 180,E1 -19438.29,E2 -19438.29} C_VEL
LIN {X 0,Y 235.588,Z 369.749,A -85,B 0,C 180,E1 -19441.709,E2 -19441.709} C_VEL
LIN {X 0,Y 235.395,Z 369.785,A -85,B 0,C 180,E1 -19446.859,E2 -19446.859} C_VEL
LIN {X 0,Y 235.228,Z 369.783,A -85,B 0,C 180,E1 -19450.327,E2 -19450.327} C_VEL
LIN {X 0,Y 235.104,Z 369.797,A -85,B 0,C 180,E1 -19455.607,E2 -19455.607} C_VEL
LIN {X 0,Y 234.999,Z 369.831,A -85,B 0,C 180,E1 -19459.206,E2 -19459.206} C_VEL
LIN {X 0,Y 234.952,Z 369.833,A -85,B 0,C 180,E1 -19462.884,E2 -19462.884} C_VEL
LIN {X 0,Y 234.955,Z 369.794,A -85,B 0,C 180,E1 -19466.659,E2 -19466.659} C_VEL
LIN {X 0,Y 234.893,Z 369.788,A -85,B 0,C 180,E1 -19470.573,E2 -19470.573} C_VEL
LIN {X 0,Y 234.952,Z 369.832,A -85,B 0,C 180,E1 -19474.634,E2 -19474.634} C_VEL
LIN {X 0,Y 234.959,Z 369.793,A -85,B 0,C 180,E1 -19478.954,E2 -19478.954} C_VEL
LIN {X 0,Y 234.991,Z 369.807,A -85,B 0,C 180,E1 -19483.462,E2 -19483.462} C_VEL
LIN {X 0,Y 235.008,Z 370.027,A -85,B 0,C 180,E1 -19484.209,E2 -19484.209} C_VEL
LIN {X 0,Y 235.705,Z 372.27,A -85,B 0,C 180,E1 -19485.335,E2 -19485.335} C_VEL
LIN {X 0,Y 238.378,Z 376.696,A -85,B 0,C 180,E1 -19486.228,E2 -19486.228} C_VEL
LIN {X 0,Y 243.3,Z 384.785,A -85,B 0,C 180,E1 -19487.647,E2 -19487.647} C_VEL
LIN {X 0,Y 250.82,Z 398.145,A -85,B 0,C 180,E1 -19489.688,E2 -19489.688} C_VEL
LIN {X 0,Y 259.189,Z 415.556,A -85,B 0,C 180,E1 -19491.845,E2 -19491.845} C_VEL
LIN {X 0,Y 264.511,Z 428.257,A -85,B 0,C 180,E1 -19493.169,E2 -19493.169} C_VEL
LIN {X 0,Y 261.502,Z 496.264,A -85,B 0,C 180,E1 -19494.941,E2 -19494.941} C_VEL
LIN {X 0,Y 260.493,Z 513.8,A -85,B 0,C 180,E1 -19495.491,E2 -19495.491} C_VEL
LIN {X 0,Y 258.899,Z 527.749,A -85,B 0,C 180,E1 -19496.19,E2 -19496.19} C_VEL
LIN {X 0,Y 256.846,Z 541.328,A -85,B 0,C 180,E1 -19497.174,E2 -19497.174} C_VEL
LIN {X 0,Y 254.6,Z 553.596,A -85,B 0,C 180,E1 -19498.37,E2 -19498.37} C_VEL
LIN {X 0,Y 251.944,Z 565.673,A -85,B 0,C 180,E1 -19499.863,E2 -19499.863} C_VEL
LIN {X 0,Y 248.951,Z 577.859,A -85,B 0,C 180,E1 -19501.783,E2 -19501.783} C_VEL
LIN {X 0,Y 246.012,Z 587.925,A -85,B 0,C 180,E1 -19503.72,E2 -19503.72} C_VEL
LIN {X 0,Y 242.976,Z 597.931,A -85,B 0,C 180,E1 -19506.115,E2 -19506.115} C_VEL
LIN {X 0,Y 240.271,Z 606.238,A -85,B 0,C 180,E1 -19508.556,E2 -19508.556} C_VEL
LIN {X 0,Y 237.87,Z 614.179,A -85,B 0,C 180,E1 -19511.484,E2 -19511.484} C_VEL
LIN {X 0,Y 235.892,Z 620.568,A -85,B 0,C 180,E1 -19514.449,E2 -19514.449} C_VEL
LIN {X 0,Y 234.522,Z 624.991,A -85,B 0,C 180,E1 -19517.014,E2 -19517.014} C_VEL
LIN {X 0,Y 233.658,Z 628.474,A -85,B 0,C 180,E1 -19519.605,E2 -19519.605} C_VEL
LIN {X 0,Y 232.92,Z 631.854,A -85,B 0,C 180,E1 -19523.07,E2 -19523.07} C_VEL
LIN {X 0,Y 232.656,Z 633.846,A -85,B 0,C 180,E1 -19526.539,E2 -19526.539} C_VEL
LIN {X 0,Y 232.687,Z 634.5,A -85,B 0,C 180,E1 -19530.002,E2 -19530.002} C_VEL
LIN {X 0,Y 232.654,Z 633.826,A -85,B 0,C 180,E1 -19533.466,E2 -19533.466} C_VEL
LIN {X 0,Y 232.893,Z 632.452,A -85,B 0,C 180,E1 -19536.282,E2 -19536.282} C_VEL
LIN {X 0,Y 233.384,Z 633.064,A -85,B 0,C 180,E1 -19538.662,E2 -19538.662} C_VEL
LIN {X 0,Y 234.686,Z 632.671,A -85,B 0,C 180,E1 -19542.102,E2 -19542.102} C_VEL
LIN {X 0,Y 235.617,Z 631.883,A -85,B 0,C 180,E1 -19543.807,E2 -19543.807} C_VEL
LIN {X 0,Y 238.164,Z 629.126,A -85,B 0,C 180,E1 -19547.165,E2 -19547.165} C_VEL
LIN {X 0,Y 241.422,Z 624.833,A -85,B 0,C 180,E1 -19550.448,E2 -19550.448} C_VEL
LIN {X 0,Y 245.72,Z 618.728,A -85,B 0,C 180,E1 -19553.607,E2 -19553.607} C_VEL
LIN {X 0,Y 250.158,Z 611.852,A -85,B 0,C 180,E1 -19556.265,E2 -19556.265} C_VEL
LIN {X 0,Y 254.347,Z 604.667,A -85,B 0,C 180,E1 -19558.468,E2 -19558.468} C_VEL
LIN {X 0,Y 259.94,Z 594.399,A -85,B 0,C 180,E1 -19560.913,E2 -19560.913} C_VEL
LIN {X 0,Y 265.137,Z 583.599,A -85,B 0,C 180,E1 -19562.917,E2 -19562.917} C_VEL
LIN {X 0,Y 269.727,Z 572.907,A -85,B 0,C 180,E1 -19564.523,E2 -19564.523} C_VEL
LIN {X 0,Y 274.762,Z 559.707,A -85,B 0,C 180,E1 -19566.039,E2 -19566.039} C_VEL
LIN {X 0,Y 278.921,Z 546.536,A -85,B 0,C 180,E1 -19567.211,E2 -19567.211} C_VEL
LIN {X 0,Y 282.498,Z 532.836,A -85,B 0,C 180,E1 -19568.12,E2 -19568.12} C_VEL
LIN {X 0,Y 289.28,Z 501.468,A -85,B 0,C 180,E1 -19569.625,E2 -19569.625} C_VEL
LIN {X 0,Y 298.65,Z 460.041,A -85,B 0,C 180,E1 -19571.479,E2 -19571.479} C_VEL
LIN {X 0,Y 297.515,Z 459.933,A -85,B 0,C 180,E1 -19573.948,E2 -19573.948} C_VEL
LIN {X 0,Y 297.201,Z 461.394,A -85,B 0,C 180,E1 -19576.176,E2 -19576.176} C_VEL
LIN {X 0,Y 297.431,Z 464.118,A -85,B 0,C 180,E1 -19578.044,E2 -19578.044} C_VEL
LIN {X 0,Y 297.675,Z 466.977,A -85,B 0,C 180,E1 -19579.25,E2 -19579.25} C_VEL
LIN {X 0,Y 296.418,Z 477.654,A -85,B 0,C 180,E1 -19580.664,E2 -19580.664} C_VEL
LIN {X 0,Y 284.519,Z 535.406,A -85,B 0,C 180,E1 -19583.312,E2 -19583.312} C_VEL
LIN {X 0,Y 280.729,Z 549.421,A -85,B 0,C 180,E1 -19584.184,E2 -19584.184} C_VEL
LIN {X 0,Y 276.776,Z 561.32,A -85,B 0,C 180,E1 -19585.157,E2 -19585.157} C_VEL
LIN {X 0,Y 271.977,Z 573.695,A -85,B 0,C 180,E1 -19586.472,E2 -19586.472} C_VEL
LIN {X 0,Y 266.559,Z 585.835,A -85,B 0,C 180,E1 -19588.176,E2 -19588.176} C_VEL
LIN {X 0,Y 261.097,Z 596.664,A -85,B 0,C 180,E1 -19590.134,E2 -19590.134} C_VEL
LIN {X 0,Y 256.127,Z 605.534,A -85,B 0,C 180,E1 -19592.195,E2 -19592.195} C_VEL
LIN {X 0,Y 251.51,Z 612.924,A -85,B 0,C 180,E1 -19594.334,E2 -19594.334} C_VEL
LIN {X 0,Y 247.455,Z 618.958,A -85,B 0,C 180,E1 -19596.571,E2 -19596.571} C_VEL
LIN {X 0,Y 243.817,Z 623.85,A -85,B 0,C 180,E1 -19598.881,E2 -19598.881} C_VEL
LIN {X 0,Y 240.853,Z 627.689,A -85,B 0,C 180,E1 -19601.278,E2 -19601.278} C_VEL
LIN {X 0,Y 237.625,Z 631.306,A -85,B 0,C 180,E1 -19604.563,E2 -19604.563} C_VEL
LIN {X 0,Y 236.31,Z 632.539,A -85,B 0,C 180,E1 -19606.236,E2 -19606.236} C_VEL
LIN {X 0,Y 235.172,Z 633.364,A -85,B 0,C 180,E1 -19607.925,E2 -19607.925} C_VEL
LIN {X 0,Y 233.629,Z 633.799,A -85,B 0,C 180,E1 -19611.349,E2 -19611.349} C_VEL
LIN {X 0,Y 232.887,Z 632.681,A -85,B 0,C 180,E1 -19614.806,E2 -19614.806} C_VEL
LIN {X 0,Y 232.793,Z 631.485,A -85,B 0,C 180,E1 -19616.539,E2 -19616.539} C_VEL
LIN {X 0,Y 232.785,Z 628.903,A -85,B 0,C 180,E1 -19619.135,E2 -19619.135} C_VEL
LIN {X 0,Y 232.87,Z 625.257,A -85,B 0,C 180,E1 -19621.73,E2 -19621.73} C_VEL
LIN {X 0,Y 233.069,Z 620.415,A -85,B 0,C 180,E1 -19624.324,E2 -19624.324} C_VEL
LIN {X 0,Y 233.264,Z 614.212,A -85,B 0,C 180,E1 -19626.922,E2 -19626.922} C_VEL
LIN {X 0,Y 233.642,Z 607.845,A -85,B 0,C 180,E1 -19629.086,E2 -19629.086} C_VEL
LIN {X 0,Y 234.147,Z 600.182,A -85,B 0,C 180,E1 -19631.251,E2 -19631.251} C_VEL
LIN {X 0,Y 234.965,Z 589.893,A -85,B 0,C 180,E1 -19633.624,E2 -19633.624} C_VEL
LIN {X 0,Y 235.965,Z 578.311,A -85,B 0,C 180,E1 -19635.77,E2 -19635.77} C_VEL
LIN {X 0,Y 237.022,Z 565.469,A -85,B 0,C 180,E1 -19637.645,E2 -19637.645} C_VEL
LIN {X 0,Y 238.028,Z 552.484,A -85,B 0,C 180,E1 -19639.116,E2 -19639.116} C_VEL
LIN {X 0,Y 238.92,Z 538.643,A -85,B 0,C 180,E1 -19640.299,E2 -19640.299} C_VEL
LIN {X 0,Y 239.607,Z 525.055,A -85,B 0,C 180,E1 -19641.114,E2 -19641.114} C_VEL
LIN {X 0,Y 242.461,Z 456.127,A -85,B 0,C 180,E1 -19644.465,E2 -19644.465} C_VEL
LIN {X 0,Y 240.039,Z 428.671,A -85,B 0,C 180,E1 -19645.917,E2 -19645.917} C_VEL
LIN {X 0,Y 239.775,Z 419.679,A -85,B 0,C 180,E1 -19646.434,E2 -19646.434} C_VEL
LIN {X 0,Y 241.879,Z 401.216,A -85,B 0,C 180,E1 -19650.563,E2 -19650.563} C_VEL
LIN {X 0,Y 238.28,Z 384.523,A -85,B 0,C 180,E1 -19654.695,E2 -19654.695} C_VEL
LIN {X 0,Y 235.036,Z 370.108,A -85,B 0,C 180,E1 -19658.432,E2 -19658.432} C_VEL
LIN {X 0,Y 234.974,Z 369.842,A -85,B 0,C 180,E1 -19658.951,E2 -19658.951} C_VEL
LIN {X 0,Y 234.916,Z 369.964,A -85,B 0,C 180,E1 -19664.261,E2 -19664.261} C_VEL
LIN {X 0,Y 235.745,Z 372.477,A -85,B 0,C 180,E1 -19665.5,E2 -19665.5} C_VEL
LIN {X 0,Y 238.658,Z 377.181,A -85,B 0,C 180,E1 -19666.425,E2 -19666.425} C_VEL
LIN {X 0,Y 246.735,Z 390.689,A -85,B 0,C 180,E1 -19668.7,E2 -19668.7} C_VEL
LIN {X 0,Y 253.99,Z 404.578,A -85,B 0,C 180,E1 -19670.624,E2 -19670.624} C_VEL
LIN {X 0,Y 261.104,Z 420.062,A -85,B 0,C 180,E1 -19672.423,E2 -19672.423} C_VEL
LIN {X 0,Y 264.327,Z 427.996,A -85,B 0,C 180,E1 -19673.223,E2 -19673.223} C_VEL
LIN {X 0,Y 261.438,Z 495.915,A -85,B 0,C 180,E1 -19675.011,E2 -19675.011} C_VEL
LIN {X 0,Y 260.46,Z 513.081,A -85,B 0,C 180,E1 -19675.54,E2 -19675.54} C_VEL
LIN {X 0,Y 258.875,Z 527.277,A -85,B 0,C 180,E1 -19676.24,E2 -19676.24} C_VEL
LIN {X 0,Y 256.919,Z 540.415,A -85,B 0,C 180,E1 -19677.18,E2 -19677.18} C_VEL
LIN {X 0,Y 254.634,Z 552.871,A -85,B 0,C 180,E1 -19678.37,E2 -19678.37} C_VEL
LIN {X 0,Y 251.971,Z 565.093,A -85,B 0,C 180,E1 -19679.862,E2 -19679.862} C_VEL
LIN {X 0,Y 249.24,Z 576.298,A -85,B 0,C 180,E1 -19681.584,E2 -19681.584} C_VEL
LIN {X 0,Y 246.049,Z 587.56,A -85,B 0,C 180,E1 -19683.72,E2 -19683.72} C_VEL
LIN {X 0,Y 243.017,Z 597.627,A -85,B 0,C 180,E1 -19686.115,E2 -19686.115} C_VEL
LIN {X 0,Y 240.349,Z 605.986,A -85,B 0,C 180,E1 -19688.559,E2 -19688.559} C_VEL
LIN {X 0,Y 237.869,Z 613.972,A -85,B 0,C 180,E1 -19691.479,E2 -19691.479} C_VEL
LIN {X 0,Y 235.903,Z 620.404,A -85,B 0,C 180,E1 -19694.445,E2 -19694.445} C_VEL
LIN {X 0,Y 234.538,Z 624.864,A -85,B 0,C 180,E1 -19697.01,E2 -19697.01} C_VEL
LIN {X 0,Y 233.665,Z 628.361,A -85,B 0,C 180,E1 -19699.601,E2 -19699.601} C_VEL
LIN {X 0,Y 232.923,Z 631.775,A -85,B 0,C 180,E1 -19703.066,E2 -19703.066} C_VEL
LIN {X 0,Y 232.655,Z 633.805,A -85,B 0,C 180,E1 -19706.534,E2 -19706.534} C_VEL
LIN {X 0,Y 232.688,Z 634.499,A -85,B 0,C 180,E1 -19709.998,E2 -19709.998} C_VEL
LIN {X 0,Y 232.654,Z 633.865,A -85,B 0,C 180,E1 -19713.461,E2 -19713.461} C_VEL
LIN {X 0,Y 232.92,Z 631.891,A -85,B 0,C 180,E1 -19716.93,E2 -19716.93} C_VEL
LIN {X 0,Y 233.657,Z 628.528,A -85,B 0,C 180,E1 -19720.395,E2 -19720.395} C_VEL
LIN {X 0,Y 234.87,Z 623.677,A -85,B 0,C 180,E1 -19723.848,E2 -19723.848} C_VEL
LIN {X 0,Y 236.42,Z 619,A -85,B 0,C 180,E1 -19726.401,E2 -19726.401} C_VEL
LIN {X 0,Y 238.461,Z 612.064,A -85,B 0,C 180,E1 -19729.418,E2 -19729.418} C_VEL
LIN {X 0,Y 241.087,Z 603.762,A -85,B 0,C 180,E1 -19732.267,E2 -19732.267} C_VEL
LIN {X 0,Y 243.867,Z 594.954,A -85,B 0,C 180,E1 -19734.698,E2 -19734.698} C_VEL
LIN {X 0,Y 247.076,Z 584.281,A -85,B 0,C 180,E1 -19737.07,E2 -19737.07} C_VEL
LIN {X 0,Y 249.893,Z 574.047,A -85,B 0,C 180,E1 -19738.909,E2 -19738.909} C_VEL
LIN {X 0,Y 252.855,Z 561.681,A -85,B 0,C 180,E1 -19740.71,E2 -19740.71} C_VEL
LIN {X 0,Y 255.562,Z 548.638,A -85,B 0,C 180,E1 -19742.193,E2 -19742.193} C_VEL
LIN {X 0,Y 257.745,Z 536.116,A -85,B 0,C 180,E1 -19743.279,E2 -19743.279} C_VEL
LIN {X 0,Y 259.557,Z 522.198,A -85,B 0,C 180,E1 -19744.181,E2 -19744.181} C_VEL
LIN {X 0,Y 260.902,Z 507.835,A -85,B 0,C 180,E1 -19744.783,E2 -19744.783} C_VEL
LIN {X 0,Y 264.493,Z 429.758,A -85,B 0,C 180,E1 -19746.829,E2 -19746.829} C_VEL
LIN {X 0,Y 264.266,Z 427.699,A -85,B 0,C 180,E1 -19746.934,E2 -19746.934} C_VEL
LIN {X 0,Y 257.275,Z 411.364,A -85,B 0,C 180,E1 -19748.682,E2 -19748.682} C_VEL
LIN {X 0,Y 249.042,Z 394.802,A -85,B 0,C 180,E1 -19750.83,E2 -19750.83} C_VEL
LIN {X 0,Y 241.276,Z 381.332,A -85,B 0,C 180,E1 -19752.976,E2 -19752.976} C_VEL
LIN {X 0,Y 235.822,Z 372.545,A -85,B 0,C 180,E1 -19754.634,E2 -19754.634} C_VEL
LIN {X 0,Y 235.099,Z 370.444,A -85,B 0,C 180,E1 -19755.579,E2 -19755.579} C_VEL
LIN {X 0,Y 234.974,Z 369.823,A -85,B 0,C 180,E1 -19756.2,E2 -19756.2} C_VEL
LIN {X 0,Y 234.962,Z 369.838,A -85,B 0,C 180,E1 -19758.849,E2 -19758.849} C_VEL
LIN {X 0,Y 234.938,Z 369.795,A -85,B 0,C 180,E1 -19763.253,E2 -19763.253} C_VEL
LIN {X 0,Y 234.952,Z 369.828,A -85,B 0,C 180,E1 -19767.423,E2 -19767.423} C_VEL
LIN {X 0,Y 234.914,Z 369.778,A -85,B 0,C 180,E1 -19771.763,E2 -19771.763} C_VEL
LIN {X 0,Y 234.981,Z 369.836,A -85,B 0,C 180,E1 -19775.246,E2 -19775.246} C_VEL
LIN {X 0,Y 234.989,Z 369.818,A -85,B 0,C 180,E1 -19779.192,E2 -19779.192} C_VEL
LIN {X 0,Y 234.284,Z 369.921,A -85,B 0,C 180,E1 -19780.623,E2 -19780.623} C_VEL
LIN {X 0,Y 231.451,Z 370.264,A -85,B 0,C 180,E1 -19782.961,E2 -19782.961} C_VEL
LIN {X 0,Y 229.092,Z 370.552,A -85,B 0,C 180,E1 -19784.867,E2 -19784.867} C_VEL
LIN {X 0,Y 228.112,Z 370.683,A -85,B 0,C 180,E1 -19786.345,E2 -19786.345} C_VEL
LIN {X 0,Y 228.047,Z 370.691,A -85,B 0,C 180,E1 -19786.845,E2 -19786.845} C_VEL
LIN {X 0,Y 228.296,Z 370.646,A -85,B 0,C 180,E1 -19791.146,E2 -19791.146} C_VEL
LIN {X 0,Y 228.346,Z 370.661,A -85,B 0,C 180,E1 -19792.928,E2 -19792.928} C_VEL
LIN {X 0,Y 228.546,Z 370.624,A -85,B 0,C 180,E1 -19798.238,E2 -19798.238} C_VEL
LIN {X 0,Y 228.546,Z 370.625,A -85,B 0,C 180,E1 -19801.762,E2 -19801.762} C_VEL
LIN {X 0,Y 228.346,Z 370.661,A -85,B 0,C 180,E1 -19807.072,E2 -19807.072} C_VEL
LIN {X 0,Y 228.154,Z 370.666,A -85,B 0,C 180,E1 -19810.651,E2 -19810.651} C_VEL
LIN {X 0,Y 228.056,Z 370.681,A -85,B 0,C 180,E1 -19814.273,E2 -19814.273} C_VEL
LIN {X 0,Y 227.994,Z 370.705,A -85,B 0,C 180,E1 -19817.954,E2 -19817.954} C_VEL
LIN {X 0,Y 227.921,Z 370.701,A -85,B 0,C 180,E1 -19822.33,E2 -19822.33} C_VEL
LIN {X 0,Y 227.931,Z 370.668,A -85,B 0,C 180,E1 -19826.602,E2 -19826.602} C_VEL
LIN {X 0,Y 227.868,Z 370.658,A -85,B 0,C 180,E1 -19830.284,E2 -19830.284} C_VEL
LIN {X 0,Y 227.881,Z 370.726,A -85,B 0,C 180,E1 -19833.72,E2 -19833.72} C_VEL
LIN {X 0,Y 227.864,Z 370.67,A -85,B 0,C 180,E1 -19838.087,E2 -19838.087} C_VEL
LIN {X 0,Y 227.966,Z 370.892,A -85,B 0,C 180,E1 -19842.781,E2 -19842.781} C_VEL
LIN {X 0,Y 228.472,Z 372.627,A -85,B 0,C 180,E1 -19843.57,E2 -19843.57} C_VEL
LIN {X 0,Y 232.568,Z 379.053,A -85,B 0,C 180,E1 -19844.94,E2 -19844.94} C_VEL
LIN {X 0,Y 237.895,Z 387.488,A -85,B 0,C 180,E1 -19846.558,E2 -19846.558} C_VEL
LIN {X 0,Y 245.468,Z 401.111,A -85,B 0,C 180,E1 -19848.732,E2 -19848.732} C_VEL
LIN {X 0,Y 252.843,Z 416.305,A -85,B 0,C 180,E1 -19850.732,E2 -19850.732} C_VEL
LIN {X 0,Y 258.772,Z 430.251,A -85,B 0,C 180,E1 -19852.279,E2 -19852.279} C_VEL
LIN {X 0,Y 255.684,Z 497.277,A -85,B 0,C 180,E1 -19854.055,E2 -19854.055} C_VEL
LIN {X 0,Y 254.689,Z 513.814,A -85,B 0,C 180,E1 -19854.589,E2 -19854.589} C_VEL
LIN {X 0,Y 253.043,Z 527.758,A -85,B 0,C 180,E1 -19855.297,E2 -19855.297} C_VEL
LIN {X 0,Y 250.915,Z 541.335,A -85,B 0,C 180,E1 -19856.296,E2 -19856.296} C_VEL
LIN {X 0,Y 248.577,Z 553.601,A -85,B 0,C 180,E1 -19857.51,E2 -19857.51} C_VEL
LIN {X 0,Y 245.678,Z 566.259,A -85,B 0,C 180,E1 -19859.115,E2 -19859.115} C_VEL
LIN {X 0,Y 242.693,Z 577.862,A -85,B 0,C 180,E1 -19860.987,E2 -19860.987} C_VEL
LIN {X 0,Y 239.664,Z 587.928,A -85,B 0,C 180,E1 -19862.968,E2 -19862.968} C_VEL
LIN {X 0,Y 236.468,Z 597.933,A -85,B 0,C 180,E1 -19865.415,E2 -19865.415} C_VEL
LIN {X 0,Y 233.635,Z 606.24,A -85,B 0,C 180,E1 -19867.916,E2 -19867.916} C_VEL
LIN {X 0,Y 231.115,Z 614.181,A -85,B 0,C 180,E1 -19870.922,E2 -19870.922} C_VEL
LIN {X 0,Y 229.033,Z 620.569,A -85,B 0,C 180,E1 -19873.971,E2 -19873.971} C_VEL
LIN {X 0,Y 227.578,Z 624.992,A -85,B 0,C 180,E1 -19876.61,E2 -19876.61} C_VEL
LIN {X 0,Y 226.637,Z 628.474,A -85,B 0,C 180,E1 -19879.279,E2 -19879.279} C_VEL
LIN {X 0,Y 225.845,Z 631.854,A -85,B 0,C 180,E1 -19882.852,E2 -19882.852} C_VEL
LIN {X 0,Y 225.57,Z 633.847,A -85,B 0,C 180,E1 -19886.43,E2 -19886.43} C_VEL
LIN {X 0,Y 225.586,Z 634.5,A -85,B 0,C 180,E1 -19890.002,E2 -19890.002} C_VEL
LIN {X 0,Y 225.571,Z 633.825,A -85,B 0,C 180,E1 -19893.575,E2 -19893.575} C_VEL
LIN {X 0,Y 225.87,Z 632.258,A -85,B 0,C 180,E1 -19896.703,E2 -19896.703} C_VEL
LIN {X 0,Y 226.345,Z 632.994,A -85,B 0,C 180,E1 -19898.933,E2 -19898.933} C_VEL
LIN {X 0,Y 227.725,Z 632.895,A -85,B 0,C 180,E1 -19902.478,E2 -19902.478} C_VEL
LIN {X 0,Y 229.959,Z 631.295,A -85,B 0,C 180,E1 -19905.968,E2 -19905.968} C_VEL
LIN {X 0,Y 233.063,Z 628.17,A -85,B 0,C 180,E1 -19909.374,E2 -19909.374} C_VEL
LIN {X 0,Y 235.994,Z 624.783,A -85,B 0,C 180,E1 -19911.857,E2 -19911.857} C_VEL
LIN {X 0,Y 239.437,Z 620.442,A -85,B 0,C 180,E1 -19914.265,E2 -19914.265} C_VEL
LIN {X 0,Y 244.781,Z 613.014,A -85,B 0,C 180,E1 -19917.349,E2 -19917.349} C_VEL
LIN {X 0,Y 250.092,Z 604.846,A -85,B 0,C 180,E1 -19919.923,E2 -19919.923} C_VEL
LIN {X 0,Y 256.088,Z 594.741,A -85,B 0,C 180,E1 -19922.356,E2 -19922.356} C_VEL
LIN {X 0,Y 261.678,Z 584.11,A -85,B 0,C 180,E1 -19924.335,E2 -19924.335} C_VEL
LIN {X 0,Y 266.587,Z 573.683,A -85,B 0,C 180,E1 -19925.916,E2 -19925.916} C_VEL
LIN {X 0,Y 271.948,Z 560.769,A -85,B 0,C 180,E1 -19927.397,E2 -19927.397} C_VEL
LIN {X 0,Y 276.367,Z 548.041,A -85,B 0,C 180,E1 -19928.54,E2 -19928.54} C_VEL
LIN {X 0,Y 280.451,Z 533.865,A -85,B 0,C 180,E1 -19929.488,E2 -19929.488} C_VEL
LIN {X 0,Y 287.683,Z 502.44,A -85,B 0,C 180,E1 -19930.981,E2 -19930.981} C_VEL
LIN {X 0,Y 296.235,Z 466.681,A -85,B 0,C 180,E1 -19932.55,E2 -19932.55} C_VEL
LIN {X 0,Y 295.493,Z 467.182,A -85,B 0,C 180,E1 -19934.708,E2 -19934.708} C_VEL
LIN {X 0,Y 295.362,Z 468.671,A -85,B 0,C 180,E1 -19936.367,E2 -19936.367} C_VEL
LIN {X 0,Y 295.434,Z 470.798,A -85,B 0,C 180,E1 -19937.712,E2 -19937.712} C_VEL
LIN {X 0,Y 295.489,Z 472.44,A -85,B 0,C 180,E1 -19938.393,E2 -19938.393} C_VEL
LIN {X 0,Y 294.268,Z 480.509,A -85,B 0,C 180,E1 -19939.45,E2 -19939.45} C_VEL
LIN {X 0,Y 282.175,Z 535.554,A -85,B 0,C 180,E1 -19941.944,E2 -19941.944} C_VEL
LIN {X 0,Y 278.512,Z 548.42,A -85,B 0,C 180,E1 -19942.727,E2 -19942.727} C_VEL
LIN {X 0,Y 273.753,Z 561.937,A -85,B 0,C 180,E1 -19943.809,E2 -19943.809} C_VEL
LIN {X 0,Y 268.702,Z 574.108,A -85,B 0,C 180,E1 -19945.1,E2 -19945.1} C_VEL
LIN {X 0,Y 262.977,Z 586.039,A -85,B 0,C 180,E1 -19946.78,E2 -19946.78} C_VEL
LIN {X 0,Y 257.18,Z 596.741,A -85,B 0,C 180,E1 -19948.72,E2 -19948.72} C_VEL
LIN {X 0,Y 251.871,Z 605.535,A -85,B 0,C 180,E1 -19950.771,E2 -19950.771} C_VEL
LIN {X 0,Y 246.899,Z 612.854,A -85,B 0,C 180,E1 -19952.907,E2 -19952.907} C_VEL
LIN {X 0,Y 242.481,Z 618.875,A -85,B 0,C 180,E1 -19955.149,E2 -19955.149} C_VEL
LIN {X 0,Y 238.496,Z 623.756,A -85,B 0,C 180,E1 -19957.475,E2 -19957.475} C_VEL
LIN {X 0,Y 235.163,Z 627.597,A -85,B 0,C 180,E1 -19959.899,E2 -19959.899} C_VEL
LIN {X 0,Y 232.428,Z 630.468,A -85,B 0,C 180,E1 -19962.4,E2 -19962.4} C_VEL
LIN {X 0,Y 229.441,Z 632.906,A -85,B 0,C 180,E1 -19965.815,E2 -19965.815} C_VEL
LIN {X 0,Y 227.313,Z 633.826,A -85,B 0,C 180,E1 -19969.309,E2 -19969.309} C_VEL
LIN {X 0,Y 226.599,Z 633.7,A -85,B 0,C 180,E1 -19971.079,E2 -19971.079} C_VEL
LIN {X 0,Y 225.829,Z 632.223,A -85,B 0,C 180,E1 -19974.643,E2 -19974.643} C_VEL
LIN {X 0,Y 225.748,Z 630.901,A -85,B 0,C 180,E1 -19976.43,E2 -19976.43} C_VEL
LIN {X 0,Y 225.733,Z 628.084,A -85,B 0,C 180,E1 -19979.108,E2 -19979.108} C_VEL
LIN {X 0,Y 225.848,Z 624.19,A -85,B 0,C 180,E1 -19981.783,E2 -19981.783} C_VEL
LIN {X 0,Y 226.036,Z 619.097,A -85,B 0,C 180,E1 -19984.458,E2 -19984.458} C_VEL
LIN {X 0,Y 226.292,Z 612.576,A -85,B 0,C 180,E1 -19987.136,E2 -19987.136} C_VEL
LIN {X 0,Y 226.739,Z 604.391,A -85,B 0,C 180,E1 -19989.816,E2 -19989.816} C_VEL
LIN {X 0,Y 227.342,Z 596.078,A -85,B 0,C 180,E1 -19992.044,E2 -19992.044} C_VEL
LIN {X 0,Y 228.161,Z 585.918,A -85,B 0,C 180,E1 -19994.266,E2 -19994.266} C_VEL
LIN {X 0,Y 229.154,Z 574.773,A -85,B 0,C 180,E1 -19996.252,E2 -19996.252} C_VEL
LIN {X 0,Y 230.143,Z 562.645,A -85,B 0,C 180,E1 -19997.975,E2 -19997.975} C_VEL
LIN {X 0,Y 231.075,Z 549.886,A -85,B 0,C 180,E1 -19999.403,E2 -19999.403} C_VEL
LIN {X 0,Y 231.98,Z 535.843,A -85,B 0,C 180,E1 -20000.563,E2 -20000.563} C_VEL
LIN {X 0,Y 232.597,Z 522.925,A -85,B 0,C 180,E1 -20001.317,E2 -20001.317} C_VEL
LIN {X 0,Y 235.439,Z 456.592,A -85,B 0,C 180,E1 -20004.688,E2 -20004.688} C_VEL
LIN {X 0,Y 233.03,Z 428.843,A -85,B 0,C 180,E1 -20006.197,E2 -20006.197} C_VEL
LIN {X 0,Y 232.782,Z 419.737,A -85,B 0,C 180,E1 -20006.727,E2 -20006.727} C_VEL
LIN {X 0,Y 234.802,Z 401.784,A -85,B 0,C 180,E1 -20010.836,E2 -20010.836} C_VEL
LIN {X 0,Y 230.897,Z 384.043,A -85,B 0,C 180,E1 -20015.333,E2 -20015.333} C_VEL
LIN {X 0,Y 227.971,Z 370.928,A -85,B 0,C 180,E1 -20018.846,E2 -20018.846} C_VEL
LIN {X 0,Y 227.852,Z 370.909,A -85,B 0,C 180,E1 -20022.884,E2 -20022.884} C_VEL
LIN {X 0,Y 228.213,Z 372.235,A -85,B 0,C 180,E1 -20023.556,E2 -20023.556} C_VEL
LIN {X 0,Y 231.13,Z 376.824,A -85,B 0,C 180,E1 -20024.605,E2 -20024.605} C_VEL
LIN {X 0,Y 237.871,Z 387.676,A -85,B 0,C 180,E1 -20026.672,E2 -20026.672} C_VEL
LIN {X 0,Y 244.633,Z 399.54,A -85,B 0,C 180,E1 -20028.606,E2 -20028.606} C_VEL
LIN {X 0,Y 252.042,Z 414.645,A -85,B 0,C 180,E1 -20030.623,E2 -20030.623} C_VEL
LIN {X 0,Y 258.436,Z 429.652,A -85,B 0,C 180,E1 -20032.297,E2 -20032.297} C_VEL
LIN {X 0,Y 258.638,Z 431.691,A -85,B 0,C 180,E1 -20032.401,E2 -20032.401} C_VEL
LIN {X 0,Y 254.931,Z 509.505,A -85,B 0,C 180,E1 -20034.492,E2 -20034.492} C_VEL
LIN {X 0,Y 253.423,Z 524.239,A -85,B 0,C 180,E1 -20035.17,E2 -20035.17} C_VEL
LIN {X 0,Y 251.327,Z 538.164,A -85,B 0,C 180,E1 -20036.113,E2 -20036.113} C_VEL
LIN {X 0,Y 248.973,Z 551.112,A -85,B 0,C 180,E1 -20037.324,E2 -20037.324} C_VEL
LIN {X 0,Y 246.175,Z 563.672,A -85,B 0,C 180,E1 -20038.837,E2 -20038.837} C_VEL
LIN {X 0,Y 243.333,Z 575.129,A -85,B 0,C 180,E1 -20040.592,E2 -20040.592} C_VEL
LIN {X 0,Y 240.262,Z 585.644,A -85,B 0,C 180,E1 -20042.565,E2 -20042.565} C_VEL
LIN {X 0,Y 237.007,Z 596.089,A -85,B 0,C 180,E1 -20045.002,E2 -20045.002} C_VEL
LIN {X 0,Y 234.157,Z 604.706,A -85,B 0,C 180,E1 -20047.498,E2 -20047.498} C_VEL
LIN {X 0,Y 231.353,Z 612.965,A -85,B 0,C 180,E1 -20050.477,E2 -20050.477} C_VEL
LIN {X 0,Y 229.631,Z 618.726,A -85,B 0,C 180,E1 -20053.095,E2 -20053.095} C_VEL
LIN {X 0,Y 227.976,Z 623.461,A -85,B 0,C 180,E1 -20055.72,E2 -20055.72} C_VEL
LIN {X 0,Y 226.644,Z 628.362,A -85,B 0,C 180,E1 -20059.275,E2 -20059.275} C_VEL
LIN {X 0,Y 225.847,Z 631.776,A -85,B 0,C 180,E1 -20062.847,E2 -20062.847} C_VEL
LIN {X 0,Y 225.573,Z 633.805,A -85,B 0,C 180,E1 -20066.425,E2 -20066.425} C_VEL
LIN {X 0,Y 225.587,Z 634.499,A -85,B 0,C 180,E1 -20069.998,E2 -20069.998} C_VEL
LIN {X 0,Y 225.572,Z 633.865,A -85,B 0,C 180,E1 -20073.57,E2 -20073.57} C_VEL
LIN {X 0,Y 225.845,Z 631.891,A -85,B 0,C 180,E1 -20077.148,E2 -20077.148} C_VEL
LIN {X 0,Y 226.636,Z 628.527,A -85,B 0,C 180,E1 -20080.721,E2 -20080.721} C_VEL
LIN {X 0,Y 227.95,Z 623.675,A -85,B 0,C 180,E1 -20084.277,E2 -20084.277} C_VEL
LIN {X 0,Y 229.581,Z 618.999,A -85,B 0,C 180,E1 -20086.904,E2 -20086.904} C_VEL
LIN {X 0,Y 231.561,Z 612.591,A -85,B 0,C 180,E1 -20089.801,E2 -20089.801} C_VEL
LIN {X 0,Y 234.06,Z 605.111,A -85,B 0,C 180,E1 -20092.507,E2 -20092.507} C_VEL
LIN {X 0,Y 236.885,Z 596.575,A -85,B 0,C 180,E1 -20095.007,E2 -20095.007} C_VEL
LIN {X 0,Y 240.147,Z 586.228,A -85,B 0,C 180,E1 -20097.445,E2 -20097.445} C_VEL
LIN {X 0,Y 243.179,Z 575.83,A -85,B 0,C 180,E1 -20099.424,E2 -20099.424} C_VEL
LIN {X 0,Y 246.092,Z 564.526,A -85,B 0,C 180,E1 -20101.17,E2 -20101.17} C_VEL
LIN {X 0,Y 248.842,Z 552.165,A -85,B 0,C 180,E1 -20102.691,E2 -20102.691} C_VEL
LIN {X 0,Y 251.191,Z 539.498,A -85,B 0,C 180,E1 -20103.903,E2 -20103.903} C_VEL
LIN {X 0,Y 253.377,Z 525.278,A -85,B 0,C 180,E1 -20104.893,E2 -20104.893} C_VEL
LIN {X 0,Y 254.871,Z 511.101,A -85,B 0,C 180,E1 -20105.572,E2 -20105.572} C_VEL
LIN {X 0,Y 256.126,Z 488.329,A -85,B 0,C 180,E1 -20106.222,E2 -20106.222} C_VEL
LIN {X 0,Y 258.727,Z 430.277,A -85,B 0,C 180,E1 -20107.772,E2 -20107.772} C_VEL
LIN {X 0,Y 252.245,Z 414.995,A -85,B 0,C 180,E1 -20109.471,E2 -20109.471} C_VEL
LIN {X 0,Y 244.402,Z 399.037,A -85,B 0,C 180,E1 -20111.612,E2 -20111.612} C_VEL
LIN {X 0,Y 237.076,Z 386.163,A -85,B 0,C 180,E1 -20113.73,E2 -20113.73} C_VEL
LIN {X 0,Y 231.019,Z 376.62,A -85,B 0,C 180,E1 -20115.597,E2 -20115.597} C_VEL
LIN {X 0,Y 228.284,Z 372.145,A -85,B 0,C 180,E1 -20116.613,E2 -20116.613} C_VEL
LIN {X 0,Y 227.934,Z 370.768,A -85,B 0,C 180,E1 -20117.434,E2 -20117.434} C_VEL
LIN {X 0,Y 227.864,Z 370.671,A -85,B 0,C 180,E1 -20121.913,E2 -20121.913} C_VEL
LIN {X 0,Y 227.884,Z 370.726,A -85,B 0,C 180,E1 -20126.371,E2 -20126.371} C_VEL
LIN {X 0,Y 227.896,Z 370.65,A -85,B 0,C 180,E1 -20130.434,E2 -20130.434} C_VEL
LIN {X 0,Y 227.921,Z 370.695,A -85,B 0,C 180,E1 -20134.425,E2 -20134.425} C_VEL
LIN {X 0,Y 227.913,Z 370.699,A -85,B 0,C 180,E1 -20139.185,E2 -20139.185} C_VEL
LIN {X 0,Y 228.048,Z 370.679,A -85,B 0,C 180,E1 -20143.897,E2 -20143.897} C_VEL
LIN {X 0,Y 228.047,Z 370.691,A -85,B 0,C 180,E1 -20146.845,E2 -20146.845} C_VEL
LIN {X 0,Y 227.432,Z 370.783,A -85,B 0,C 180,E1 -20148.321,E2 -20148.321} C_VEL
LIN {X 0,Y 224.654,Z 371.143,A -85,B 0,C 180,E1 -20150.732,E2 -20150.732} C_VEL
LIN {X 0,Y 221.457,Z 371.527,A -85,B 0,C 180,E1 -20153.711,E2 -20153.711} C_VEL
LIN {X 0,Y 221.134,Z 371.553,A -85,B 0,C 180,E1 -20154.741,E2 -20154.741} C_VEL
LIN {X 0,Y 221.504,Z 371.5,A -85,B 0,C 180,E1 -20158.182,E2 -20158.182} C_VEL
LIN {X 0,Y 221.504,Z 371.5,A -85,B 0,C 180,E1 -20161.818,E2 -20161.818} C_VEL
LIN {X 0,Y 221.297,Z 371.537,A -85,B 0,C 180,E1 -20167.298,E2 -20167.298} C_VEL
LIN {X 0,Y 221.103,Z 371.547,A -85,B 0,C 180,E1 -20170.994,E2 -20170.994} C_VEL
LIN {X 0,Y 221.007,Z 371.556,A -85,B 0,C 180,E1 -20176.63,E2 -20176.63} C_VEL
LIN {X 0,Y 220.883,Z 371.574,A -85,B 0,C 180,E1 -20180.487,E2 -20180.487} C_VEL
LIN {X 0,Y 220.858,Z 371.597,A -85,B 0,C 180,E1 -20184.436,E2 -20184.436} C_VEL
LIN {X 0,Y 220.804,Z 371.53,A -85,B 0,C 180,E1 -20188.518,E2 -20188.518} C_VEL
LIN {X 0,Y 220.811,Z 371.587,A -85,B 0,C 180,E1 -20192.757,E2 -20192.757} C_VEL
LIN {X 0,Y 220.83,Z 371.546,A -85,B 0,C 180,E1 -20197.289,E2 -20197.289} C_VEL
LIN {X 0,Y 220.867,Z 371.801,A -85,B 0,C 180,E1 -20201.104,E2 -20201.104} C_VEL
LIN {X 0,Y 221.097,Z 372.716,A -85,B 0,C 180,E1 -20201.522,E2 -20201.522} C_VEL
LIN {X 0,Y 222.634,Z 375.446,A -85,B 0,C 180,E1 -20202.146,E2 -20202.146} C_VEL
LIN {X 0,Y 224.613,Z 377.795,A -85,B 0,C 180,E1 -20202.809,E2 -20202.809} C_VEL
LIN {X 0,Y 231.334,Z 388.346,A -85,B 0,C 180,E1 -20205.034,E2 -20205.034} C_VEL
LIN {X 0,Y 238.025,Z 399.881,A -85,B 0,C 180,E1 -20207.09,E2 -20207.09} C_VEL
LIN {X 0,Y 244.649,Z 412.961,A -85,B 0,C 180,E1 -20209.017,E2 -20209.017} C_VEL
LIN {X 0,Y 251.319,Z 427.941,A -85,B 0,C 180,E1 -20210.869,E2 -20210.869} C_VEL
LIN {X 0,Y 253.047,Z 432.292,A -85,B 0,C 180,E1 -20211.342,E2 -20211.342} C_VEL
LIN {X 0,Y 250.216,Z 493.16,A -85,B 0,C 180,E1 -20212.996,E2 -20212.996} C_VEL
LIN {X 0,Y 249.104,Z 512.179,A -85,B 0,C 180,E1 -20213.579,E2 -20213.579} C_VEL
LIN {X 0,Y 247.5,Z 526.244,A -85,B 0,C 180,E1 -20214.278,E2 -20214.278} C_VEL
LIN {X 0,Y 245.22,Z 540.213,A -85,B 0,C 180,E1 -20215.279,E2 -20215.279} C_VEL
LIN {X 0,Y 242.607,Z 553.607,A -85,B 0,C 180,E1 -20216.608,E2 -20216.608} C_VEL
LIN {X 0,Y 239.758,Z 565.682,A -85,B 0,C 180,E1 -20218.157,E2 -20218.157} C_VEL
LIN {X 0,Y 236.497,Z 577.865,A -85,B 0,C 180,E1 -20220.151,E2 -20220.151} C_VEL
LIN {X 0,Y 233.348,Z 587.931,A -85,B 0,C 180,E1 -20222.174,E2 -20222.174} C_VEL
LIN {X 0,Y 229.994,Z 597.935,A -85,B 0,C 180,E1 -20224.675,E2 -20224.675} C_VEL
LIN {X 0,Y 227.045,Z 606.242,A -85,B 0,C 180,E1 -20227.239,E2 -20227.239} C_VEL
LIN {X 0,Y 224.374,Z 614.182,A -85,B 0,C 180,E1 -20230.325,E2 -20230.325} C_VEL
LIN {X 0,Y 222.193,Z 620.57,A -85,B 0,C 180,E1 -20233.463,E2 -20233.463} C_VEL
LIN {X 0,Y 220.255,Z 626.235,A -85,B 0,C 180,E1 -20237.096,E2 -20237.096} C_VEL
LIN {X 0,Y 219.136,Z 630.344,A -85,B 0,C 180,E1 -20240.775,E2 -20240.775} C_VEL
LIN {X 0,Y 218.595,Z 633.02,A -85,B 0,C 180,E1 -20244.467,E2 -20244.467} C_VEL
LIN {X 0,Y 218.472,Z 634.339,A -85,B 0,C 180,E1 -20248.159,E2 -20248.159} C_VEL
LIN {X 0,Y 218.488,Z 634.5,A -85,B 0,C 180,E1 -20250.002,E2 -20250.002} C_VEL
LIN {X 0,Y 218.498,Z 633.825,A -85,B 0,C 180,E1 -20253.691,E2 -20253.691} C_VEL
LIN {X 0,Y 218.902,Z 632.116,A -85,B 0,C 180,E1 -20257.381,E2 -20257.381} C_VEL
LIN {X 0,Y 219.935,Z 633.126,A -85,B 0,C 180,E1 -20261.056,E2 -20261.056} C_VEL
LIN {X 0,Y 221.864,Z 632.654,A -85,B 0,C 180,E1 -20264.682,E2 -20264.682} C_VEL
LIN {X 0,Y 224.69,Z 630.646,A -85,B 0,C 180,E1 -20268.229,E2 -20268.229} C_VEL
LIN {X 0,Y 228.357,Z 627.183,A -85,B 0,C 180,E1 -20271.676,E2 -20271.676} C_VEL
LIN {X 0,Y 233.151,Z 622.069,A -85,B 0,C 180,E1 -20274.964,E2 -20274.964} C_VEL
LIN {X 0,Y 238.788,Z 615.237,A -85,B 0,C 180,E1 -20278.096,E2 -20278.096} C_VEL
LIN {X 0,Y 243.505,Z 608.838,A -85,B 0,C 180,E1 -20280.339,E2 -20280.339} C_VEL
LIN {X 0,Y 249.699,Z 599.728,A -85,B 0,C 180,E1 -20282.809,E2 -20282.809} C_VEL
LIN {X 0,Y 255.444,Z 590.329,A -85,B 0,C 180,E1 -20284.815,E2 -20284.815} C_VEL
LIN {X 0,Y 262.098,Z 577.962,A -85,B 0,C 180,E1 -20286.87,E2 -20286.87} C_VEL
LIN {X 0,Y 267.654,Z 566.133,A -85,B 0,C 180,E1 -20288.343,E2 -20288.343} C_VEL
LIN {X 0,Y 272.862,Z 553.24,A -85,B 0,C 180,E1 -20289.606,E2 -20289.606} C_VEL
LIN {X 0,Y 277.725,Z 538.587,A -85,B 0,C 180,E1 -20290.666,E2 -20290.666} C_VEL
LIN {X 0,Y 282.249,Z 520.72,A -85,B 0,C 180,E1 -20291.587,E2 -20291.587} C_VEL
LIN {X 0,Y 293.97,Z 473.617,A -85,B 0,C 180,E1 -20293.656,E2 -20293.656} C_VEL
LIN {X 0,Y 293.568,Z 474.755,A -85,B 0,C 180,E1 -20295.55,E2 -20295.55} C_VEL
LIN {X 0,Y 293.492,Z 476.913,A -85,B 0,C 180,E1 -20297.122,E2 -20297.122} C_VEL
LIN {X 0,Y 293.397,Z 478.014,A -85,B 0,C 180,E1 -20297.542,E2 -20297.542} C_VEL
LIN {X 0,Y 292.497,Z 483.042,A -85,B 0,C 180,E1 -20298.174,E2 -20298.174} C_VEL
LIN {X 0,Y 280.414,Z 535.051,A -85,B 0,C 180,E1 -20300.508,E2 -20300.508} C_VEL
LIN {X 0,Y 276.582,Z 547.877,A -85,B 0,C 180,E1 -20301.265,E2 -20301.265} C_VEL
LIN {X 0,Y 272.186,Z 559.928,A -85,B 0,C 180,E1 -20302.176,E2 -20302.176} C_VEL
LIN {X 0,Y 266.831,Z 572.301,A -85,B 0,C 180,E1 -20303.422,E2 -20303.422} C_VEL
LIN {X 0,Y 261.798,Z 582.497,A -85,B 0,C 180,E1 -20304.748,E2 -20304.748} C_VEL
LIN {X 0,Y 256.488,Z 592.04,A -85,B 0,C 180,E1 -20306.298,E2 -20306.298} C_VEL
LIN {X 0,Y 250.532,Z 601.573,A -85,B 0,C 180,E1 -20308.266,E2 -20308.266} C_VEL
LIN {X 0,Y 245.113,Z 609.483,A -85,B 0,C 180,E1 -20310.357,E2 -20310.357} C_VEL
LIN {X 0,Y 240.844,Z 615.047,A -85,B 0,C 180,E1 -20312.167,E2 -20312.167} C_VEL
LIN {X 0,Y 236.237,Z 620.603,A -85,B 0,C 180,E1 -20314.445,E2 -20314.445} C_VEL
LIN {X 0,Y 232.081,Z 625.117,A -85,B 0,C 180,E1 -20316.817,E2 -20316.817} C_VEL
LIN {X 0,Y 229.651,Z 627.552,A -85,B 0,C 180,E1 -20318.455,E2 -20318.455} C_VEL
LIN {X 0,Y 225.724,Z 631.147,A -85,B 0,C 180,E1 -20321.859,E2 -20321.859} C_VEL
LIN {X 0,Y 222.572,Z 633.251,A -85,B 0,C 180,E1 -20325.368,E2 -20325.368} C_VEL
LIN {X 0,Y 220.328,Z 633.782,A -85,B 0,C 180,E1 -20328.966,E2 -20328.966} C_VEL
LIN {X 0,Y 219.093,Z 632.799,A -85,B 0,C 180,E1 -20332.628,E2 -20332.628} C_VEL
LIN {X 0,Y 218.749,Z 631.418,A -85,B 0,C 180,E1 -20334.876,E2 -20334.876} C_VEL
LIN {X 0,Y 218.715,Z 628.302,A -85,B 0,C 180,E1 -20338.159,E2 -20338.159} C_VEL
LIN {X 0,Y 218.78,Z 624.524,A -85,B 0,C 180,E1 -20340.92,E2 -20340.92} C_VEL
LIN {X 0,Y 218.975,Z 619.577,A -85,B 0,C 180,E1 -20343.681,E2 -20343.681} C_VEL
LIN {X 0,Y 219.181,Z 613.705,A -85,B 0,C 180,E1 -20346.258,E2 -20346.258} C_VEL
LIN {X 0,Y 219.543,Z 606.752,A -85,B 0,C 180,E1 -20348.746,E2 -20348.746} C_VEL
LIN {X 0,Y 220.175,Z 597.143,A -85,B 0,C 180,E1 -20351.508,E2 -20351.508} C_VEL
LIN {X 0,Y 220.96,Z 587.322,A -85,B 0,C 180,E1 -20353.801,E2 -20353.801} C_VEL
LIN {X 0,Y 221.883,Z 576.481,A -85,B 0,C 180,E1 -20355.854,E2 -20355.854} C_VEL
LIN {X 0,Y 222.873,Z 564.67,A -85,B 0,C 180,E1 -20357.669,E2 -20357.669} C_VEL
LIN {X 0,Y 223.912,Z 551.108,A -85,B 0,C 180,E1 -20359.281,E2 -20359.281} C_VEL
LIN {X 0,Y 224.812,Z 536.961,A -85,B 0,C 180,E1 -20360.531,E2 -20360.531} C_VEL
LIN {X 0,Y 225.499,Z 523.686,A -85,B 0,C 180,E1 -20361.362,E2 -20361.362} C_VEL
LIN {X 0,Y 228.362,Z 456.809,A -85,B 0,C 180,E1 -20364.913,E2 -20364.913} C_VEL
LIN {X 0,Y 226.028,Z 428.628,A -85,B 0,C 180,E1 -20366.514,E2 -20366.514} C_VEL
LIN {X 0,Y 225.836,Z 419.611,A -85,B 0,C 180,E1 -20367.067,E2 -20367.067} C_VEL
LIN {X 0,Y 227.692,Z 403.971,A -85,B 0,C 180,E1 -20370.719,E2 -20370.719} C_VEL
LIN {X 0,Y 227.145,Z 399.911,A -85,B 0,C 180,E1 -20371.735,E2 -20371.735} C_VEL
LIN {X 0,Y 223.351,Z 382.519,A -85,B 0,C 180,E1 -20376.276,E2 -20376.276} C_VEL
LIN {X 0,Y 220.881,Z 371.822,A -85,B 0,C 180,E1 -20379.24,E2 -20379.24} C_VEL
LIN {X 0,Y 220.774,Z 371.749,A -85,B 0,C 180,E1 -20381.17,E2 -20381.17} C_VEL
LIN {X 0,Y 221.024,Z 372.802,A -85,B 0,C 180,E1 -20381.653,E2 -20381.653} C_VEL
LIN {X 0,Y 222.579,Z 375.518,A -85,B 0,C 180,E1 -20382.263,E2 -20382.263} C_VEL
LIN {X 0,Y 224.547,Z 377.883,A -85,B 0,C 180,E1 -20382.923,E2 -20382.923} C_VEL
LIN {X 0,Y 228.786,Z 384.439,A -85,B 0,C 180,E1 -20384.342,E2 -20384.342} C_VEL
LIN {X 0,Y 233.95,Z 392.955,A -85,B 0,C 180,E1 -20385.98,E2 -20385.98} C_VEL
LIN {X 0,Y 238.978,Z 401.854,A -85,B 0,C 180,E1 -20387.492,E2 -20387.492} C_VEL
LIN {X 0,Y 245.318,Z 414.453,A -85,B 0,C 180,E1 -20389.314,E2 -20389.314} C_VEL
LIN {X 0,Y 252.335,Z 430.508,A -85,B 0,C 180,E1 -20391.248,E2 -20391.248} C_VEL
LIN {X 0,Y 253.014,Z 432.344,A -85,B 0,C 180,E1 -20391.436,E2 -20391.436} C_VEL
LIN {X 0,Y 249.176,Z 509.655,A -85,B 0,C 180,E1 -20393.55,E2 -20393.55} C_VEL
LIN {X 0,Y 247.639,Z 524.249,A -85,B 0,C 180,E1 -20394.234,E2 -20394.234} C_VEL
LIN {X 0,Y 245.457,Z 538.172,A -85,B 0,C 180,E1 -20395.188,E2 -20395.188} C_VEL
LIN {X 0,Y 243.027,Z 551.118,A -85,B 0,C 180,E1 -20396.42,E2 -20396.42} C_VEL
LIN {X 0,Y 240.114,Z 563.677,A -85,B 0,C 180,E1 -20397.958,E2 -20397.958} C_VEL
LIN {X 0,Y 237.164,Z 575.133,A -85,B 0,C 180,E1 -20399.748,E2 -20399.748} C_VEL
LIN {X 0,Y 233.972,Z 585.647,A -85,B 0,C 180,E1 -20401.762,E2 -20401.762} C_VEL
LIN {X 0,Y 230.556,Z 596.092,A -85,B 0,C 180,E1 -20404.252,E2 -20404.252} C_VEL
LIN {X 0,Y 227.577,Z 604.708,A -85,B 0,C 180,E1 -20406.81,E2 -20406.81} C_VEL
LIN {X 0,Y 224.607,Z 612.966,A -85,B 0,C 180,E1 -20409.865,E2 -20409.865} C_VEL
LIN {X 0,Y 222.809,Z 618.728,A -85,B 0,C 180,E1 -20412.561,E2 -20412.561} C_VEL
LIN {X 0,Y 221.076,Z 623.462,A -85,B 0,C 180,E1 -20415.265,E2 -20415.265} C_VEL
LIN {X 0,Y 219.648,Z 628.363,A -85,B 0,C 180,E1 -20418.929,E2 -20418.929} C_VEL
LIN {X 0,Y 218.798,Z 631.777,A -85,B 0,C 180,E1 -20422.616,E2 -20422.616} C_VEL
LIN {X 0,Y 218.5,Z 633.805,A -85,B 0,C 180,E1 -20426.309,E2 -20426.309} C_VEL
LIN {X 0,Y 218.489,Z 634.499,A -85,B 0,C 180,E1 -20429.998,E2 -20429.998} C_VEL
LIN {X 0,Y 218.498,Z 633.865,A -85,B 0,C 180,E1 -20433.686,E2 -20433.686} C_VEL
LIN {X 0,Y 218.796,Z 631.89,A -85,B 0,C 180,E1 -20437.38,E2 -20437.38} C_VEL
LIN {X 0,Y 219.639,Z 628.527,A -85,B 0,C 180,E1 -20441.066,E2 -20441.066} C_VEL
LIN {X 0,Y 221.051,Z 623.674,A -85,B 0,C 180,E1 -20444.732,E2 -20444.732} C_VEL
LIN {X 0,Y 222.762,Z 618.997,A -85,B 0,C 180,E1 -20447.438,E2 -20447.438} C_VEL
LIN {X 0,Y 224.686,Z 613.067,A -85,B 0,C 180,E1 -20450.219,E2 -20450.219} C_VEL
LIN {X 0,Y 227.496,Z 605.109,A -85,B 0,C 180,E1 -20453.194,E2 -20453.194} C_VEL
LIN {X 0,Y 230.454,Z 596.572,A -85,B 0,C 180,E1 -20455.755,E2 -20455.755} C_VEL
LIN {X 0,Y 233.861,Z 586.225,A -85,B 0,C 180,E1 -20458.247,E2 -20458.247} C_VEL
LIN {X 0,Y 237.003,Z 575.826,A -85,B 0,C 180,E1 -20460.27,E2 -20460.27} C_VEL
LIN {X 0,Y 240.042,Z 564.522,A -85,B 0,C 180,E1 -20462.048,E2 -20462.048} C_VEL
LIN {X 0,Y 242.896,Z 552.16,A -85,B 0,C 180,E1 -20463.595,E2 -20463.595} C_VEL
LIN {X 0,Y 245.332,Z 539.49,A -85,B 0,C 180,E1 -20464.827,E2 -20464.827} C_VEL
LIN {X 0,Y 247.444,Z 526.029,A -85,B 0,C 180,E1 -20465.794,E2 -20465.794} C_VEL
LIN {X 0,Y 249.122,Z 511.256,A -85,B 0,C 180,E1 -20466.514,E2 -20466.514} C_VEL
LIN {X 0,Y 250.371,Z 489.775,A -85,B 0,C 180,E1 -20467.141,E2 -20467.141} C_VEL
LIN {X 0,Y 253.037,Z 432.208,A -85,B 0,C 180,E1 -20468.708,E2 -20468.708} C_VEL
LIN {X 0,Y 246.443,Z 416.831,A -85,B 0,C 180,E1 -20470.521,E2 -20470.521} C_VEL
LIN {X 0,Y 239.707,Z 403.114,A -85,B 0,C 180,E1 -20472.454,E2 -20472.454} C_VEL
LIN {X 0,Y 232.918,Z 390.942,A -85,B 0,C 180,E1 -20474.513,E2 -20474.513} C_VEL
LIN {X 0,Y 226.675,Z 381.034,A -85,B 0,C 180,E1 -20476.529,E2 -20476.529} C_VEL
LIN {X 0,Y 223.396,Z 376.196,A -85,B 0,C 180,E1 -20477.649,E2 -20477.649} C_VEL
LIN {X 0,Y 221.465,Z 373.711,A -85,B 0,C 180,E1 -20478.327,E2 -20478.327} C_VEL
LIN {X 0,Y 220.935,Z 372.108,A -85,B 0,C 180,E1 -20478.735,E2 -20478.735} C_VEL
LIN {X 0,Y 220.864,Z 371.598,A -85,B 0,C 180,E1 -20479.479,E2 -20479.479} C_VEL
LIN {X 0,Y 220.827,Z 371.547,A -85,B 0,C 180,E1 -20482.793,E2 -20482.793} C_VEL
LIN {X 0,Y 220.816,Z 371.589,A -85,B 0,C 180,E1 -20487.243,E2 -20487.243} C_VEL
LIN {X 0,Y 220.819,Z 371.529,A -85,B 0,C 180,E1 -20491.484,E2 -20491.484} C_VEL
LIN {X 0,Y 220.86,Z 371.597,A -85,B 0,C 180,E1 -20495.564,E2 -20495.564} C_VEL
LIN {X 0,Y 220.884,Z 371.575,A -85,B 0,C 180,E1 -20499.513,E2 -20499.513} C_VEL
LIN {X 0,Y 221.007,Z 371.559,A -85,B 0,C 180,E1 -20503.369,E2 -20503.369} C_VEL
LIN {X 0,Y 221.103,Z 371.549,A -85,B 0,C 180,E1 -20509.005,E2 -20509.005} C_VEL
LIN {X 0,Y 221.297,Z 371.536,A -85,B 0,C 180,E1 -20512.702,E2 -20512.702} C_VEL
LIN {X 0,Y 221.134,Z 371.553,A -85,B 0,C 180,E1 -20514.741,E2 -20514.741} C_VEL
LIN {X 0,Y 220.506,Z 371.621,A -85,B 0,C 180,E1 -20516.267,E2 -20516.267} C_VEL
LIN {X 0,Y 217.845,Z 371.964,A -85,B 0,C 180,E1 -20518.766,E2 -20518.766} C_VEL
LIN {X 0,Y 214.668,Z 372.354,A -85,B 0,C 180,E1 -20521.846,E2 -20521.846} C_VEL
LIN {X 0,Y 214.242,Z 372.396,A -85,B 0,C 180,E1 -20522.91,E2 -20522.91} C_VEL
LIN {X 0,Y 214.231,Z 372.412,A -85,B 0,C 180,E1 -20527.54,E2 -20527.54} C_VEL
LIN {X 0,Y 214.035,Z 372.432,A -85,B 0,C 180,E1 -20531.362,E2 -20531.362} C_VEL
LIN {X 0,Y 213.924,Z 372.434,A -85,B 0,C 180,E1 -20535.237,E2 -20535.237} C_VEL
LIN {X 0,Y 213.831,Z 372.466,A -85,B 0,C 180,E1 -20539.188,E2 -20539.188} C_VEL
LIN {X 0,Y 213.838,Z 372.465,A -85,B 0,C 180,E1 -20543.228,E2 -20543.228} C_VEL
LIN {X 0,Y 213.802,Z 372.41,A -85,B 0,C 180,E1 -20547.442,E2 -20547.442} C_VEL
LIN {X 0,Y 213.752,Z 372.437,A -85,B 0,C 180,E1 -20551.74,E2 -20551.74} C_VEL
LIN {X 0,Y 213.746,Z 372.436,A -85,B 0,C 180,E1 -20556.288,E2 -20556.288} C_VEL
LIN {X 0,Y 213.824,Z 372.632,A -85,B 0,C 180,E1 -20558.947,E2 -20558.947} C_VEL
LIN {X 0,Y 214.078,Z 373.661,A -85,B 0,C 180,E1 -20559.423,E2 -20559.423} C_VEL
LIN {X 0,Y 215.659,Z 376.404,A -85,B 0,C 180,E1 -20560.102,E2 -20560.102} C_VEL
LIN {X 0,Y 217.414,Z 378.149,A -85,B 0,C 180,E1 -20560.736,E2 -20560.736} C_VEL
LIN {X 0,Y 219.568,Z 381.41,A -85,B 0,C 180,E1 -20561.542,E2 -20561.542} C_VEL
LIN {X 0,Y 221.257,Z 383.641,A -85,B 0,C 180,E1 -20562.14,E2 -20562.14} C_VEL
LIN {X 0,Y 227.283,Z 393.187,A -85,B 0,C 180,E1 -20564.219,E2 -20564.219} C_VEL
LIN {X 0,Y 233.679,Z 404.45,A -85,B 0,C 180,E1 -20566.281,E2 -20566.281} C_VEL
LIN {X 0,Y 240.178,Z 417.461,A -85,B 0,C 180,E1 -20568.26,E2 -20568.26} C_VEL
LIN {X 0,Y 247.106,Z 433.429,A -85,B 0,C 180,E1 -20570.272,E2 -20570.272} C_VEL
LIN {X 0,Y 247.52,Z 434.534,A -85,B 0,C 180,E1 -20570.393,E2 -20570.393} C_VEL
LIN {X 0,Y 244.314,Z 498.15,A -85,B 0,C 180,E1 -20572.127,E2 -20572.127} C_VEL
LIN {X 0,Y 243.257,Z 513.841,A -85,B 0,C 180,E1 -20572.651,E2 -20572.651} C_VEL
LIN {X 0,Y 241.508,Z 527.776,A -85,B 0,C 180,E1 -20573.379,E2 -20573.379} C_VEL
LIN {X 0,Y 239.217,Z 541.348,A -85,B 0,C 180,E1 -20574.406,E2 -20574.406} C_VEL
LIN {X 0,Y 236.695,Z 553.612,A -85,B 0,C 180,E1 -20575.66,E2 -20575.66} C_VEL
LIN {X 0,Y 233.74,Z 565.686,A -85,B 0,C 180,E1 -20577.236,E2 -20577.236} C_VEL
LIN {X 0,Y 230.359,Z 577.868,A -85,B 0,C 180,E1 -20579.271,E2 -20579.271} C_VEL
LIN {X 0,Y 227.071,Z 587.933,A -85,B 0,C 180,E1 -20581.335,E2 -20581.335} C_VEL
LIN {X 0,Y 223.569,Z 597.937,A -85,B 0,C 180,E1 -20583.893,E2 -20583.893} C_VEL
LIN {X 0,Y 220.484,Z 606.244,A -85,B 0,C 180,E1 -20586.522,E2 -20586.522} C_VEL
LIN {X 0,Y 217.662,Z 614.094,A -85,B 0,C 180,E1 -20589.648,E2 -20589.648} C_VEL
LIN {X 0,Y 215.374,Z 620.571,A -85,B 0,C 180,E1 -20592.924,E2 -20592.924} C_VEL
LIN {X 0,Y 213.291,Z 626.236,A -85,B 0,C 180,E1 -20596.667,E2 -20596.667} C_VEL
LIN {X 0,Y 212.102,Z 630.344,A -85,B 0,C 180,E1 -20600.466,E2 -20600.466} C_VEL
LIN {X 0,Y 211.508,Z 633.021,A -85,B 0,C 180,E1 -20604.281,E2 -20604.281} C_VEL
LIN {X 0,Y 211.378,Z 634.339,A -85,B 0,C 180,E1 -20608.097,E2 -20608.097} C_VEL
LIN {X 0,Y 211.392,Z 634.5,A -85,B 0,C 180,E1 -20610.002,E2 -20610.002} C_VEL
LIN {X 0,Y 211.417,Z 633.825,A -85,B 0,C 180,E1 -20613.814,E2 -20613.814} C_VEL
LIN {X 0,Y 211.909,Z 631.837,A -85,B 0,C 180,E1 -20617.865,E2 -20617.865} C_VEL
LIN {X 0,Y 212.958,Z 633.065,A -85,B 0,C 180,E1 -20621.423,E2 -20621.423} C_VEL
LIN {X 0,Y 214.984,Z 632.913,A -85,B 0,C 180,E1 -20625.163,E2 -20625.163} C_VEL
LIN {X 0,Y 217.977,Z 631.324,A -85,B 0,C 180,E1 -20628.812,E2 -20628.812} C_VEL
LIN {X 0,Y 221.87,Z 628.269,A -85,B 0,C 180,E1 -20632.343,E2 -20632.343} C_VEL
LIN {X 0,Y 226.89,Z 623.632,A -85,B 0,C 180,E1 -20635.702,E2 -20635.702} C_VEL
LIN {X 0,Y 231.273,Z 619.092,A -85,B 0,C 180,E1 -20638.102,E2 -20638.102} C_VEL
LIN {X 0,Y 236.896,Z 612.551,A -85,B 0,C 180,E1 -20640.783,E2 -20640.783} C_VEL
LIN {X 0,Y 243.259,Z 604.373,A -85,B 0,C 180,E1 -20643.296,E2 -20643.296} C_VEL
LIN {X 0,Y 249.174,Z 595.911,A -85,B 0,C 180,E1 -20645.327,E2 -20645.327} C_VEL
LIN {X 0,Y 255.482,Z 585.882,A -85,B 0,C 180,E1 -20647.245,E2 -20647.245} C_VEL
LIN {X 0,Y 261.07,Z 575.902,A -85,B 0,C 180,E1 -20648.75,E2 -20648.75} C_VEL
LIN {X 0,Y 267.032,Z 563.822,A -85,B 0,C 180,E1 -20650.154,E2 -20650.154} C_VEL
LIN {X 0,Y 271.946,Z 552.088,A -85,B 0,C 180,E1 -20651.226,E2 -20651.226} C_VEL
LIN {X 0,Y 276.752,Z 538.344,A -85,B 0,C 180,E1 -20652.174,E2 -20652.174} C_VEL
LIN {X 0,Y 281.555,Z 520.451,A -85,B 0,C 180,E1 -20653.059,E2 -20653.059} C_VEL
LIN {X 0,Y 291.818,Z 481.052,A -85,B 0,C 180,E1 -20654.752,E2 -20654.752} C_VEL
LIN {X 0,Y 291.605,Z 482.92,A -85,B 0,C 180,E1 -20656.441,E2 -20656.441} C_VEL
LIN {X 0,Y 291.551,Z 483.402,A -85,B 0,C 180,E1 -20656.625,E2 -20656.625} C_VEL
LIN {X 0,Y 291.008,Z 485.857,A -85,B 0,C 180,E1 -20656.89,E2 -20656.89} C_VEL
LIN {X 0,Y 278.56,Z 536.292,A -85,B 0,C 180,E1 -20659.126,E2 -20659.126} C_VEL
LIN {X 0,Y 274.26,Z 549.713,A -85,B 0,C 180,E1 -20659.922,E2 -20659.922} C_VEL
LIN {X 0,Y 269.672,Z 561.241,A -85,B 0,C 180,E1 -20660.803,E2 -20660.803} C_VEL
LIN {X 0,Y 264.071,Z 573.337,A -85,B 0,C 180,E1 -20662.015,E2 -20662.015} C_VEL
LIN {X 0,Y 258.769,Z 583.245,A -85,B 0,C 180,E1 -20663.309,E2 -20663.309} C_VEL
LIN {X 0,Y 253.164,Z 592.608,A -85,B 0,C 180,E1 -20664.828,E2 -20664.828} C_VEL
LIN {X 0,Y 246.904,Z 601.962,A -85,B 0,C 180,E1 -20666.774,E2 -20666.774} C_VEL
LIN {X 0,Y 241.122,Z 609.711,A -85,B 0,C 180,E1 -20668.845,E2 -20668.845} C_VEL
LIN {X 0,Y 236.52,Z 615.235,A -85,B 0,C 180,E1 -20670.641,E2 -20670.641} C_VEL
LIN {X 0,Y 231.571,Z 620.709,A -85,B 0,C 180,E1 -20672.92,E2 -20672.92} C_VEL
LIN {X 0,Y 227.077,Z 625.153,A -85,B 0,C 180,E1 -20675.303,E2 -20675.303} C_VEL
LIN {X 0,Y 223.136,Z 628.607,A -85,B 0,C 180,E1 -20677.793,E2 -20677.793} C_VEL
LIN {X 0,Y 219.021,Z 631.798,A -85,B 0,C 180,E1 -20681.284,E2 -20681.284} C_VEL
LIN {X 0,Y 215.701,Z 633.479,A -85,B 0,C 180,E1 -20684.891,E2 -20684.891} C_VEL
LIN {X 0,Y 213.364,Z 633.692,A -85,B 0,C 180,E1 -20688.601,E2 -20688.601} C_VEL
LIN {X 0,Y 212.061,Z 632.343,A -85,B 0,C 180,E1 -20692.382,E2 -20692.382} C_VEL
LIN {X 0,Y 211.659,Z 629.457,A -85,B 0,C 180,E1 -20696.192,E2 -20696.192} C_VEL
LIN {X 0,Y 211.691,Z 626.148,A -85,B 0,C 180,E1 -20699.049,E2 -20699.049} C_VEL
LIN {X 0,Y 211.849,Z 621.74,A -85,B 0,C 180,E1 -20701.901,E2 -20701.901} C_VEL
LIN {X 0,Y 212.066,Z 616.049,A -85,B 0,C 180,E1 -20704.753,E2 -20704.753} C_VEL
LIN {X 0,Y 212.383,Z 608.836,A -85,B 0,C 180,E1 -20707.606,E2 -20707.606} C_VEL
LIN {X 0,Y 212.909,Z 599.832,A -85,B 0,C 180,E1 -20710.46,E2 -20710.46} C_VEL
LIN {X 0,Y 213.688,Z 589.563,A -85,B 0,C 180,E1 -20713.068,E2 -20713.068} C_VEL
LIN {X 0,Y 214.659,Z 578.068,A -85,B 0,C 180,E1 -20715.427,E2 -20715.427} C_VEL
LIN {X 0,Y 215.745,Z 565.008,A -85,B 0,C 180,E1 -20717.537,E2 -20717.537} C_VEL
LIN {X 0,Y 216.816,Z 551.276,A -85,B 0,C 180,E1 -20719.242,E2 -20719.242} C_VEL
LIN {X 0,Y 217.699,Z 537.306,A -85,B 0,C 180,E1 -20720.536,E2 -20720.536} C_VEL
LIN {X 0,Y 218.435,Z 523.052,A -85,B 0,C 180,E1 -20721.468,E2 -20721.468} C_VEL
LIN {X 0,Y 221.359,Z 457.605,A -85,B 0,C 180,E1 -20725.096,E2 -20725.096} C_VEL
LIN {X 0,Y 219.049,Z 429.901,A -85,B 0,C 180,E1 -20726.723,E2 -20726.723} C_VEL
LIN {X 0,Y 218.825,Z 419.631,A -85,B 0,C 180,E1 -20727.366,E2 -20727.366} C_VEL
LIN {X 0,Y 220.656,Z 403.8,A -85,B 0,C 180,E1 -20731.17,E2 -20731.17} C_VEL
LIN {X 0,Y 217.342,Z 388.284,A -85,B 0,C 180,E1 -20735.264,E2 -20735.264} C_VEL
LIN {X 0,Y 214.362,Z 374.791,A -85,B 0,C 180,E1 -20739.051,E2 -20739.051} C_VEL
LIN {X 0,Y 214.295,Z 374.379,A -85,B 0,C 180,E1 -20739.451,E2 -20739.451} C_VEL
LIN {X 0,Y 214.544,Z 374.94,A -85,B 0,C 180,E1 -20739.777,E2 -20739.777} C_VEL
LIN {X 0,Y 216.654,Z 377.404,A -85,B 0,C 180,E1 -20740.602,E2 -20740.602} C_VEL
LIN {X 0,Y 217.544,Z 378.626,A -85,B 0,C 180,E1 -20740.936,E2 -20740.936} C_VEL
LIN {X 0,Y 219.859,Z 381.846,A -85,B 0,C 180,E1 -20741.782,E2 -20741.782} C_VEL
LIN {X 0,Y 224.571,Z 388.932,A -85,B 0,C 180,E1 -20743.435,E2 -20743.435} C_VEL
LIN {X 0,Y 230.332,Z 398.578,A -85,B 0,C 180,E1 -20745.345,E2 -20745.345} C_VEL
LIN {X 0,Y 236.126,Z 409.248,A -85,B 0,C 180,E1 -20747.155,E2 -20747.155} C_VEL
LIN {X 0,Y 243.07,Z 423.96,A -85,B 0,C 180,E1 -20749.221,E2 -20749.221} C_VEL
LIN {X 0,Y 247.294,Z 434.023,A -85,B 0,C 180,E1 -20750.433,E2 -20750.433} C_VEL
LIN {X 0,Y 244.364,Z 495.401,A -85,B 0,C 180,E1 -20752.137,E2 -20752.137} C_VEL
LIN {X 0,Y 243.19,Z 513.127,A -85,B 0,C 180,E1 -20752.698,E2 -20752.698} C_VEL
LIN {X 0,Y 241.462,Z 527.308,A -85,B 0,C 180,E1 -20753.431,E2 -20753.431} C_VEL
LIN {X 0,Y 239.295,Z 540.437,A -85,B 0,C 180,E1 -20754.414,E2 -20754.414} C_VEL
LIN {X 0,Y 236.748,Z 552.889,A -85,B 0,C 180,E1 -20755.663,E2 -20755.663} C_VEL
LIN {X 0,Y 233.745,Z 565.107,A -85,B 0,C 180,E1 -20757.232,E2 -20757.232} C_VEL
LIN {X 0,Y 230.367,Z 577.433,A -85,B 0,C 180,E1 -20759.267,E2 -20759.267} C_VEL
LIN {X 0,Y 227.12,Z 587.569,A -85,B 0,C 180,E1 -20761.336,E2 -20761.336} C_VEL
LIN {X 0,Y 223.604,Z 597.634,A -85,B 0,C 180,E1 -20763.892,E2 -20763.892} C_VEL
LIN {X 0,Y 220.563,Z 605.993,A -85,B 0,C 180,E1 -20766.526,E2 -20766.526} C_VEL
LIN {X 0,Y 217.787,Z 613.292,A -85,B 0,C 180,E1 -20769.364,E2 -20769.364} C_VEL
LIN {X 0,Y 216.009,Z 618.729,A -85,B 0,C 180,E1 -20771.993,E2 -20771.993} C_VEL
LIN {X 0,Y 214.198,Z 623.463,A -85,B 0,C 180,E1 -20774.78,E2 -20774.78} C_VEL
LIN {X 0,Y 212.667,Z 628.364,A -85,B 0,C 180,E1 -20778.561,E2 -20778.561} C_VEL
LIN {X 0,Y 211.728,Z 631.777,A -85,B 0,C 180,E1 -20782.368,E2 -20782.368} C_VEL
LIN {X 0,Y 211.418,Z 633.806,A -85,B 0,C 180,E1 -20786.186,E2 -20786.186} C_VEL
LIN {X 0,Y 211.393,Z 634.499,A -85,B 0,C 180,E1 -20789.998,E2 -20789.998} C_VEL
LIN {X 0,Y 211.417,Z 633.864,A -85,B 0,C 180,E1 -20793.81,E2 -20793.81} C_VEL
LIN {X 0,Y 211.726,Z 631.89,A -85,B 0,C 180,E1 -20797.628,E2 -20797.628} C_VEL
LIN {X 0,Y 212.658,Z 628.526,A -85,B 0,C 180,E1 -20801.434,E2 -20801.434} C_VEL
LIN {X 0,Y 214.174,Z 623.673,A -85,B 0,C 180,E1 -20805.217,E2 -20805.217} C_VEL
LIN {X 0,Y 215.95,Z 618.996,A -85,B 0,C 180,E1 -20808.007,E2 -20808.007} C_VEL
LIN {X 0,Y 218.331,Z 612.199,A -85,B 0,C 180,E1 -20811.229,E2 -20811.229} C_VEL
LIN {X 0,Y 221.438,Z 603.755,A -85,B 0,C 180,E1 -20814.365,E2 -20814.365} C_VEL
LIN {X 0,Y 224.629,Z 594.946,A -85,B 0,C 180,E1 -20816.976,E2 -20816.976} C_VEL
LIN {X 0,Y 227.619,Z 586.222,A -85,B 0,C 180,E1 -20819.095,E2 -20819.095} C_VEL
LIN {X 0,Y 231.296,Z 574.567,A -85,B 0,C 180,E1 -20821.371,E2 -20821.371} C_VEL
LIN {X 0,Y 234.396,Z 563.092,A -85,B 0,C 180,E1 -20823.172,E2 -20823.172} C_VEL
LIN {X 0,Y 237.396,Z 550.387,A -85,B 0,C 180,E1 -20824.739,E2 -20824.739} C_VEL
LIN {X 0,Y 240.01,Z 537.223,A -85,B 0,C 180,E1 -20825.975,E2 -20825.975} C_VEL
LIN {X 0,Y 242.045,Z 523.734,A -85,B 0,C 180,E1 -20826.916,E2 -20826.916} C_VEL
LIN {X 0,Y 243.661,Z 508.96,A -85,B 0,C 180,E1 -20827.598,E2 -20827.598} C_VEL
LIN {X 0,Y 247.301,Z 438.91,A -85,B 0,C 180,E1 -20829.533,E2 -20829.533} C_VEL
LIN {X 0,Y 247.334,Z 434.049,A -85,B 0,C 180,E1 -20829.706,E2 -20829.706} C_VEL
LIN {X 0,Y 241.229,Z 419.829,A -85,B 0,C 180,E1 -20831.471,E2 -20831.471} C_VEL
LIN {X 0,Y 235.162,Z 407.347,A -85,B 0,C 180,E1 -20833.3,E2 -20833.3} C_VEL
LIN {X 0,Y 228.88,Z 395.832,A -85,B 0,C 180,E1 -20835.301,E2 -20835.301} C_VEL
LIN {X 0,Y 221.718,Z 384.329,A -85,B 0,C 180,E1 -20837.741,E2 -20837.741} C_VEL
LIN {X 0,Y 219.78,Z 381.623,A -85,B 0,C 180,E1 -20838.43,E2 -20838.43} C_VEL
LIN {X 0,Y 217.607,Z 378.533,A -85,B 0,C 180,E1 -20839.231,E2 -20839.231} C_VEL
LIN {X 0,Y 216.562,Z 377.236,A -85,B 0,C 180,E1 -20839.618,E2 -20839.618} C_VEL
LIN {X 0,Y 214.67,Z 375.049,A -85,B 0,C 180,E1 -20840.327,E2 -20840.327} C_VEL
LIN {X 0,Y 213.898,Z 373.016,A -85,B 0,C 180,E1 -20840.841,E2 -20840.841} C_VEL
LIN {X 0,Y 213.798,Z 372.51,A -85,B 0,C 180,E1 -20841.349,E2 -20841.349} C_VEL
LIN {X 0,Y 213.763,Z 372.482,A -85,B 0,C 180,E1 -20846.019,E2 -20846.019} C_VEL
LIN {X 0,Y 213.752,Z 372.409,A -85,B 0,C 180,E1 -20850.449,E2 -20850.449} C_VEL
LIN {X 0,Y 213.793,Z 372.457,A -85,B 0,C 180,E1 -20854.7,E2 -20854.7} C_VEL
LIN {X 0,Y 213.804,Z 372.455,A -85,B 0,C 180,E1 -20858.802,E2 -20858.802} C_VEL
LIN {X 0,Y 213.935,Z 372.446,A -85,B 0,C 180,E1 -20862.803,E2 -20862.803} C_VEL
LIN {X 0,Y 213.972,Z 372.449,A -85,B 0,C 180,E1 -20866.708,E2 -20866.708} C_VEL
LIN {X 0,Y 214.158,Z 372.404,A -85,B 0,C 180,E1 -20870.556,E2 -20870.556} C_VEL
LIN {X 0,Y 214.231,Z 372.411,A -85,B 0,C 180,E1 -20872.46,E2 -20872.46} C_VEL
LIN {X 0,Y 214.437,Z 372.379,A -85,B 0,C 180,E1 -20878.122,E2 -20878.122} C_VEL
LIN {X 0,Y 214.55,Z 372.385,A -85,B 0,C 180,E1 -20880,E2 -20880} C_VEL
LIN {X 0,Y 214.242,Z 372.396,A -85,B 0,C 180,E1 -20882.91,E2 -20882.91} C_VEL
LIN {X 0,Y 213.417,Z 372.505,A -85,B 0,C 180,E1 -20884.478,E2 -20884.478} C_VEL
LIN {X 0,Y 210.527,Z 372.881,A -85,B 0,C 180,E1 -20887.041,E2 -20887.041} C_VEL
LIN {X 0,Y 207.336,Z 373.258,A -85,B 0,C 180,E1 -20890.211,E2 -20890.211} C_VEL
LIN {X 0,Y 206.99,Z 373.307,A -85,B 0,C 180,E1 -20891.309,E2 -20891.309} C_VEL
LIN {X 0,Y 206.857,Z 373.313,A -85,B 0,C 180,E1 -20895.771,E2 -20895.771} C_VEL
LIN {X 0,Y 206.775,Z 373.335,A -85,B 0,C 180,E1 -20899.87,E2 -20899.87} C_VEL
LIN {X 0,Y 206.754,Z 373.356,A -85,B 0,C 180,E1 -20904.073,E2 -20904.073} C_VEL
LIN {X 0,Y 206.719,Z 373.283,A -85,B 0,C 180,E1 -20908.422,E2 -20908.422} C_VEL
LIN {X 0,Y 206.694,Z 373.345,A -85,B 0,C 180,E1 -20912.958,E2 -20912.958} C_VEL
LIN {X 0,Y 206.736,Z 373.506,A -85,B 0,C 180,E1 -20916.505,E2 -20916.505} C_VEL
LIN {X 0,Y 206.938,Z 374.457,A -85,B 0,C 180,E1 -20916.995,E2 -20916.995} C_VEL
LIN {X 0,Y 208.407,Z 377.066,A -85,B 0,C 180,E1 -20917.708,E2 -20917.708} C_VEL
LIN {X 0,Y 210.506,Z 378.96,A -85,B 0,C 180,E1 -20918.543,E2 -20918.543} C_VEL
LIN {X 0,Y 212.512,Z 382.174,A -85,B 0,C 180,E1 -20919.386,E2 -20919.386} C_VEL
LIN {X 0,Y 214.241,Z 384.191,A -85,B 0,C 180,E1 -20920.049,E2 -20920.049} C_VEL
LIN {X 0,Y 218.213,Z 389.816,A -85,B 0,C 180,E1 -20921.549,E2 -20921.549} C_VEL
LIN {X 0,Y 225.37,Z 401.544,A -85,B 0,C 180,E1 -20924.093,E2 -20924.093} C_VEL
LIN {X 0,Y 232.834,Z 415.744,A -85,B 0,C 180,E1 -20926.553,E2 -20926.553} C_VEL
LIN {X 0,Y 239.865,Z 431.414,A -85,B 0,C 180,E1 -20928.74,E2 -20928.74} C_VEL
LIN {X 0,Y 241.982,Z 436.63,A -85,B 0,C 180,E1 -20929.378,E2 -20929.378} C_VEL
LIN {X 0,Y 238.766,Z 498.112,A -85,B 0,C 180,E1 -20931.082,E2 -20931.082} C_VEL
LIN {X 0,Y 237.659,Z 513.855,A -85,B 0,C 180,E1 -20931.613,E2 -20931.613} C_VEL
LIN {X 0,Y 235.851,Z 527.785,A -85,B 0,C 180,E1 -20932.351,E2 -20932.351} C_VEL
LIN {X 0,Y 233.498,Z 541.355,A -85,B 0,C 180,E1 -20933.396,E2 -20933.396} C_VEL
LIN {X 0,Y 230.867,Z 553.617,A -85,B 0,C 180,E1 -20934.665,E2 -20934.665} C_VEL
LIN {X 0,Y 227.802,Z 565.69,A -85,B 0,C 180,E1 -20936.27,E2 -20936.27} C_VEL
LIN {X 0,Y 224.28,Z 577.872,A -85,B 0,C 180,E1 -20938.343,E2 -20938.343} C_VEL
LIN {X 0,Y 220.837,Z 587.936,A -85,B 0,C 180,E1 -20940.447,E2 -20940.447} C_VEL
LIN {X 0,Y 217.201,Z 597.94,A -85,B 0,C 180,E1 -20943.067,E2 -20943.067} C_VEL
LIN {X 0,Y 213.975,Z 606.246,A -85,B 0,C 180,E1 -20945.763,E2 -20945.763} C_VEL
LIN {X 0,Y 211.126,Z 613.643,A -85,B 0,C 180,E1 -20948.759,E2 -20948.759} C_VEL
LIN {X 0,Y 208.576,Z 620.573,A -85,B 0,C 180,E1 -20952.349,E2 -20952.349} C_VEL
LIN {X 0,Y 206.342,Z 626.237,A -85,B 0,C 180,E1 -20956.209,E2 -20956.209} C_VEL
LIN {X 0,Y 205.089,Z 630.345,A -85,B 0,C 180,E1 -20960.137,E2 -20960.137} C_VEL
LIN {X 0,Y 204.438,Z 633.021,A -85,B 0,C 180,E1 -20964.083,E2 -20964.083} C_VEL
LIN {X 0,Y 204.287,Z 634.34,A -85,B 0,C 180,E1 -20968.031,E2 -20968.031} C_VEL
LIN {X 0,Y 204.298,Z 634.5,A -85,B 0,C 180,E1 -20970.002,E2 -20970.002} C_VEL
LIN {X 0,Y 204.336,Z 633.824,A -85,B 0,C 180,E1 -20973.947,E2 -20973.947} C_VEL
LIN {X 0,Y 204.929,Z 631.519,A -85,B 0,C 180,E1 -20978.383,E2 -20978.383} C_VEL
LIN {X 0,Y 205.984,Z 632.866,A -85,B 0,C 180,E1 -20981.815,E2 -20981.815} C_VEL
LIN {X 0,Y 208.12,Z 633.119,A -85,B 0,C 180,E1 -20985.676,E2 -20985.676} C_VEL
LIN {X 0,Y 211.289,Z 631.913,A -85,B 0,C 180,E1 -20989.431,E2 -20989.431} C_VEL
LIN {X 0,Y 215.396,Z 629.276,A -85,B 0,C 180,E1 -20993.053,E2 -20993.053} C_VEL
LIN {X 0,Y 220.665,Z 625.174,A -85,B 0,C 180,E1 -20996.483,E2 -20996.483} C_VEL
LIN {X 0,Y 226.873,Z 619.428,A -85,B 0,C 180,E1 -20999.714,E2 -20999.714} C_VEL
LIN {X 0,Y 232.96,Z 613.016,A -85,B 0,C 180,E1 -21002.379,E2 -21002.379} C_VEL
LIN {X 0,Y 239.785,Z 605.037,A -85,B 0,C 180,E1 -21004.86,E2 -21004.86} C_VEL
LIN {X 0,Y 246.059,Z 596.812,A -85,B 0,C 180,E1 -21006.858,E2 -21006.858} C_VEL
LIN {X 0,Y 252.75,Z 587.077,A -85,B 0,C 180,E1 -21008.731,E2 -21008.731} C_VEL
LIN {X 0,Y 259.071,Z 576.655,A -85,B 0,C 180,E1 -21010.291,E2 -21010.291} C_VEL
LIN {X 0,Y 265.857,Z 563.802,A -85,B 0,C 180,E1 -21011.749,E2 -21011.749} C_VEL
LIN {X 0,Y 270.831,Z 552.695,A -85,B 0,C 180,E1 -21012.729,E2 -21012.729} C_VEL
LIN {X 0,Y 276.106,Z 538.533,A -85,B 0,C 180,E1 -21013.667,E2 -21013.667} C_VEL
LIN {X 0,Y 281.233,Z 520.486,A -85,B 0,C 180,E1 -21014.523,E2 -21014.523} C_VEL
LIN {X 0,Y 288.682,Z 493.138,A -85,B 0,C 180,E1 -21015.677,E2 -21015.677} C_VEL
LIN {X 0,Y 288.741,Z 492.966,A -85,B 0,C 180,E1 -21015.762,E2 -21015.762} C_VEL
LIN {X 0,Y 277.483,Z 536.313,A -85,B 0,C 180,E1 -21017.659,E2 -21017.659} C_VEL
LIN {X 0,Y 272.864,Z 549.979,A -85,B 0,C 180,E1 -21018.435,E2 -21018.435} C_VEL
LIN {X 0,Y 267.366,Z 562.899,A -85,B 0,C 180,E1 -21019.415,E2 -21019.415} C_VEL
LIN {X 0,Y 261.523,Z 574.613,A -85,B 0,C 180,E1 -21020.589,E2 -21020.589} C_VEL
LIN {X 0,Y 254.79,Z 586.189,A -85,B 0,C 180,E1 -21022.14,E2 -21022.14} C_VEL
LIN {X 0,Y 248.949,Z 595.035,A -85,B 0,C 180,E1 -21023.641,E2 -21023.641} C_VEL
LIN {X 0,Y 241.334,Z 605.226,A -85,B 0,C 180,E1 -21025.904,E2 -21025.904} C_VEL
LIN {X 0,Y 234.366,Z 613.449,A -85,B 0,C 180,E1 -21028.347,E2 -21028.347} C_VEL
LIN {X 0,Y 228.846,Z 619.204,A -85,B 0,C 180,E1 -21030.569,E2 -21030.569} C_VEL
LIN {X 0,Y 223.842,Z 623.913,A -85,B 0,C 180,E1 -21032.919,E2 -21032.919} C_VEL
LIN {X 0,Y 219.34,Z 627.642,A -85,B 0,C 180,E1 -21035.384,E2 -21035.384} C_VEL
LIN {X 0,Y 216.644,Z 629.596,A -85,B 0,C 180,E1 -21037.09,E2 -21037.09} C_VEL
LIN {X 0,Y 212.324,Z 632.359,A -85,B 0,C 180,E1 -21040.67,E2 -21040.67} C_VEL
LIN {X 0,Y 208.853,Z 633.666,A -85,B 0,C 180,E1 -21044.383,E2 -21044.383} C_VEL
LIN {X 0,Y 206.417,Z 633.47,A -85,B 0,C 180,E1 -21048.212,E2 -21048.212} C_VEL
LIN {X 0,Y 205.052,Z 631.818,A -85,B 0,C 180,E1 -21052.12,E2 -21052.12} C_VEL
LIN {X 0,Y 204.627,Z 628.569,A -85,B 0,C 180,E1 -21056.061,E2 -21056.061} C_VEL
LIN {X 0,Y 204.679,Z 625.005,A -85,B 0,C 180,E1 -21059.016,E2 -21059.016} C_VEL
LIN {X 0,Y 204.866,Z 620.311,A -85,B 0,C 180,E1 -21061.966,E2 -21061.966} C_VEL
LIN {X 0,Y 205.1,Z 614.288,A -85,B 0,C 180,E1 -21064.914,E2 -21064.914} C_VEL
LIN {X 0,Y 205.458,Z 606.739,A -85,B 0,C 180,E1 -21067.864,E2 -21067.864} C_VEL
LIN {X 0,Y 205.976,Z 597.201,A -85,B 0,C 180,E1 -21070.817,E2 -21070.817} C_VEL
LIN {X 0,Y 206.763,Z 587.531,A -85,B 0,C 180,E1 -21073.264,E2 -21073.264} C_VEL
LIN {X 0,Y 207.747,Z 575.495,A -85,B 0,C 180,E1 -21075.702,E2 -21075.702} C_VEL
LIN {X 0,Y 208.739,Z 563.493,A -85,B 0,C 180,E1 -21077.639,E2 -21077.639} C_VEL
LIN {X 0,Y 209.767,Z 550.202,A -85,B 0,C 180,E1 -21079.321,E2 -21079.321} C_VEL
LIN {X 0,Y 210.735,Z 535.322,A -85,B 0,C 180,E1 -21080.709,E2 -21080.709} C_VEL
LIN {X 0,Y 211.42,Z 521.045,A -85,B 0,C 180,E1 -21081.64,E2 -21081.64} C_VEL
LIN {X 0,Y 214.31,Z 457.939,A -85,B 0,C 180,E1 -21085.3,E2 -21085.3} C_VEL
LIN {X 0,Y 212.033,Z 430.381,A -85,B 0,C 180,E1 -21086.979,E2 -21086.979} C_VEL
LIN {X 0,Y 211.843,Z 419.6,A -85,B 0,C 180,E1 -21087.675,E2 -21087.675} C_VEL
LIN {X 0,Y 213.602,Z 404.485,A -85,B 0,C 180,E1 -21091.389,E2 -21091.389} C_VEL
LIN {X 0,Y 209.988,Z 387.817,A -85,B 0,C 180,E1 -21095.93,E2 -21095.93} C_VEL
LIN {X 0,Y 208.801,Z 382.281,A -85,B 0,C 180,E1 -21097.552,E2 -21097.552} C_VEL
LIN {X 0,Y 208.841,Z 381.711,A -85,B 0,C 180,E1 -21098.069,E2 -21098.069} C_VEL
LIN {X 0,Y 210.133,Z 382.469,A -85,B 0,C 180,E1 -21098.752,E2 -21098.752} C_VEL
LIN {X 0,Y 212.105,Z 382.278,A -85,B 0,C 180,E1 -21099.401,E2 -21099.401} C_VEL
LIN {X 0,Y 212.566,Z 382.343,A -85,B 0,C 180,E1 -21099.556,E2 -21099.556} C_VEL
LIN {X 0,Y 214.048,Z 384.059,A -85,B 0,C 180,E1 -21100.122,E2 -21100.122} C_VEL
LIN {X 0,Y 216.835,Z 387.839,A -85,B 0,C 180,E1 -21101.175,E2 -21101.175} C_VEL
LIN {X 0,Y 222.785,Z 397.273,A -85,B 0,C 180,E1 -21103.333,E2 -21103.333} C_VEL
LIN {X 0,Y 229.79,Z 409.846,A -85,B 0,C 180,E1 -21105.696,E2 -21105.696} C_VEL
LIN {X 0,Y 236.127,Z 422.967,A -85,B 0,C 180,E1 -21107.71,E2 -21107.71} C_VEL
LIN {X 0,Y 241.817,Z 436.314,A -85,B 0,C 180,E1 -21109.439,E2 -21109.439} C_VEL
LIN {X 0,Y 238.086,Z 507.499,A -85,B 0,C 180,E1 -21111.446,E2 -21111.446} C_VEL
LIN {X 0,Y 236.597,Z 521.9,A -85,B 0,C 180,E1 -21112.081,E2 -21112.081} C_VEL
LIN {X 0,Y 234.362,Z 535.928,A -85,B 0,C 180,E1 -21113.011,E2 -21113.011} C_VEL
LIN {X 0,Y 231.718,Z 549.365,A -85,B 0,C 180,E1 -21114.276,E2 -21114.276} C_VEL
LIN {X 0,Y 228.561,Z 562.261,A -85,B 0,C 180,E1 -21115.861,E2 -21115.861} C_VEL
LIN {X 0,Y 225.378,Z 573.799,A -85,B 0,C 180,E1 -21117.683,E2 -21117.683} C_VEL
LIN {X 0,Y 222.232,Z 583.703,A -85,B 0,C 180,E1 -21119.6,E2 -21119.6} C_VEL
LIN {X 0,Y 218.987,Z 592.844,A -85,B 0,C 180,E1 -21121.744,E2 -21121.744} C_VEL
LIN {X 0,Y 215.609,Z 602.006,A -85,B 0,C 180,E1 -21124.41,E2 -21124.41} C_VEL
LIN {X 0,Y 212.144,Z 610.755,A -85,B 0,C 180,E1 -21127.603,E2 -21127.603} C_VEL
LIN {X 0,Y 209.85,Z 616.922,A -85,B 0,C 180,E1 -21130.431,E2 -21130.431} C_VEL
LIN {X 0,Y 207.953,Z 622.022,A -85,B 0,C 180,E1 -21133.303,E2 -21133.303} C_VEL
LIN {X 0,Y 206,Z 627.302,A -85,B 0,C 180,E1 -21137.185,E2 -21137.185} C_VEL
LIN {X 0,Y 205.094,Z 630.25,A -85,B 0,C 180,E1 -21140.132,E2 -21140.132} C_VEL
LIN {X 0,Y 204.441,Z 632.961,A -85,B 0,C 180,E1 -21144.078,E2 -21144.078} C_VEL
LIN {X 0,Y 204.289,Z 634.318,A -85,B 0,C 180,E1 -21148.026,E2 -21148.026} C_VEL
LIN {X 0,Y 204.3,Z 634.499,A -85,B 0,C 180,E1 -21149.998,E2 -21149.998} C_VEL
LIN {X 0,Y 204.336,Z 633.864,A -85,B 0,C 180,E1 -21153.942,E2 -21153.942} C_VEL
LIN {X 0,Y 204.67,Z 631.889,A -85,B 0,C 180,E1 -21157.892,E2 -21157.892} C_VEL
LIN {X 0,Y 205.653,Z 628.525,A -85,B 0,C 180,E1 -21161.829,E2 -21161.829} C_VEL
LIN {X 0,Y 207.318,Z 623.672,A -85,B 0,C 180,E1 -21165.733,E2 -21165.733} C_VEL
LIN {X 0,Y 209.153,Z 618.994,A -85,B 0,C 180,E1 -21168.613,E2 -21168.613} C_VEL
LIN {X 0,Y 211.683,Z 612.197,A -85,B 0,C 180,E1 -21171.929,E2 -21171.929} C_VEL
LIN {X 0,Y 214.973,Z 603.753,A -85,B 0,C 180,E1 -21175.148,E2 -21175.148} C_VEL
LIN {X 0,Y 218.281,Z 594.943,A -85,B 0,C 180,E1 -21177.828,E2 -21177.828} C_VEL
LIN {X 0,Y 222.102,Z 584.268,A -85,B 0,C 180,E1 -21180.414,E2 -21180.414} C_VEL
LIN {X 0,Y 225.43,Z 574.083,A -85,B 0,C 180,E1 -21182.392,E2 -21182.392} C_VEL
LIN {X 0,Y 228.473,Z 563.087,A -85,B 0,C 180,E1 -21184.148,E2 -21184.148} C_VEL
LIN {X 0,Y 231.586,Z 550.381,A -85,B 0,C 180,E1 -21185.742,E2 -21185.742} C_VEL
LIN {X 0,Y 234.31,Z 537.216,A -85,B 0,C 180,E1 -21186.993,E2 -21186.993} C_VEL
LIN {X 0,Y 236.41,Z 523.724,A -85,B 0,C 180,E1 -21187.949,E2 -21187.949} C_VEL
LIN {X 0,Y 238.05,Z 509.296,A -85,B 0,C 180,E1 -21188.626,E2 -21188.626} C_VEL
LIN {X 0,Y 241.812,Z 440.02,A -85,B 0,C 180,E1 -21190.571,E2 -21190.571} C_VEL
LIN {X 0,Y 241.774,Z 436.109,A -85,B 0,C 180,E1 -21190.729,E2 -21190.729} C_VEL
LIN {X 0,Y 236.197,Z 423.028,A -85,B 0,C 180,E1 -21192.429,E2 -21192.429} C_VEL
LIN {X 0,Y 230.647,Z 411.449,A -85,B 0,C 180,E1 -21194.191,E2 -21194.191} C_VEL
LIN {X 0,Y 224.572,Z 400.26,A -85,B 0,C 180,E1 -21196.221,E2 -21196.221} C_VEL
LIN {X 0,Y 218.033,Z 389.534,A -85,B 0,C 180,E1 -21198.563,E2 -21198.563} C_VEL
LIN {X 0,Y 216.243,Z 387.023,A -85,B 0,C 180,E1 -21199.227,E2 -21199.227} C_VEL
LIN {X 0,Y 213.35,Z 383.033,A -85,B 0,C 180,E1 -21200.341,E2 -21200.341} C_VEL
LIN {X 0,Y 211.03,Z 380.006,A -85,B 0,C 180,E1 -21201.268,E2 -21201.268} C_VEL
LIN {X 0,Y 210.125,Z 378.559,A -85,B 0,C 180,E1 -21201.654,E2 -21201.654} C_VEL
LIN {X 0,Y 207.718,Z 376.175,A -85,B 0,C 180,E1 -21202.634,E2 -21202.634} C_VEL
LIN {X 0,Y 206.8,Z 373.881,A -85,B 0,C 180,E1 -21203.28,E2 -21203.28} C_VEL
LIN {X 0,Y 206.7,Z 373.353,A -85,B 0,C 180,E1 -21204.091,E2 -21204.091} C_VEL
LIN {X 0,Y 206.712,Z 373.314,A -85,B 0,C 180,E1 -21208.203,E2 -21208.203} C_VEL
LIN {X 0,Y 206.756,Z 373.282,A -85,B 0,C 180,E1 -21212.096,E2 -21212.096} C_VEL
LIN {X 0,Y 206.778,Z 373.349,A -85,B 0,C 180,E1 -21216.582,E2 -21216.582} C_VEL
LIN {X 0,Y 206.865,Z 373.335,A -85,B 0,C 180,E1 -21222.196,E2 -21222.196} C_VEL
LIN {X 0,Y 206.905,Z 373.321,A -85,B 0,C 180,E1 -21226.245,E2 -21226.245} C_VEL
LIN {X 0,Y 207.096,Z 373.284,A -85,B 0,C 180,E1 -21230.231,E2 -21230.231} C_VEL
LIN {X 0,Y 207.169,Z 373.286,A -85,B 0,C 180,E1 -21232.201,E2 -21232.201} C_VEL
LIN {X 0,Y 207.374,Z 373.257,A -85,B 0,C 180,E1 -21238.058,E2 -21238.058} C_VEL
LIN {X 0,Y 207.514,Z 373.262,A -85,B 0,C 180,E1 -21240,E2 -21240} C_VEL
LIN {X 0,Y 207.078,Z 373.289,A -85,B 0,C 180,E1 -21243.892,E2 -21243.892} C_VEL
LIN {X 0,Y 207.169,Z 373.286,A -85,B 0,C 180,E1 -21247.799,E2 -21247.799} C_VEL
LIN {X 0,Y 206.99,Z 373.307,A -85,B 0,C 180,E1 -21251.309,E2 -21251.309} C_VEL
LIN {X 0,Y 206.249,Z 373.417,A -85,B 0,C 180,E1 -21252.931,E2 -21252.931} C_VEL
LIN {X 0,Y 203.306,Z 373.789,A -85,B 0,C 180,E1 -21255.578,E2 -21255.578} C_VEL
LIN {X 0,Y 200.833,Z 374.086,A -85,B 0,C 180,E1 -21257.744,E2 -21257.744} C_VEL
LIN {X 0,Y 199.774,Z 374.212,A -85,B 0,C 180,E1 -21259.429,E2 -21259.429} C_VEL
LIN {X 0,Y 199.686,Z 374.214,A -85,B 0,C 180,E1 -21260.001,E2 -21260.001} C_VEL
LIN {X 0,Y 199.728,Z 374.23,A -85,B 0,C 180,E1 -21263.818,E2 -21263.818} C_VEL
LIN {X 0,Y 199.69,Z 374.157,A -85,B 0,C 180,E1 -21268.381,E2 -21268.381} C_VEL
LIN {X 0,Y 199.664,Z 374.249,A -85,B 0,C 180,E1 -21273.214,E2 -21273.214} C_VEL
LIN {X 0,Y 199.722,Z 374.725,A -85,B 0,C 180,E1 -21273.998,E2 -21273.998} C_VEL
LIN {X 0,Y 200.512,Z 376.798,A -85,B 0,C 180,E1 -21274.666,E2 -21274.666} C_VEL
LIN {X 0,Y 202.608,Z 379.132,A -85,B 0,C 180,E1 -21275.654,E2 -21275.654} C_VEL
LIN {X 0,Y 203.596,Z 379.891,A -85,B 0,C 180,E1 -21276.085,E2 -21276.085} C_VEL
LIN {X 0,Y 205.628,Z 383.154,A -85,B 0,C 180,E1 -21277.041,E2 -21277.041} C_VEL
LIN {X 0,Y 207.564,Z 385.225,A -85,B 0,C 180,E1 -21277.858,E2 -21277.858} C_VEL
LIN {X 0,Y 210.11,Z 388.74,A -85,B 0,C 180,E1 -21278.931,E2 -21278.931} C_VEL
LIN {X 0,Y 214.573,Z 394.989,A -85,B 0,C 180,E1 -21280.7,E2 -21280.7} C_VEL
LIN {X 0,Y 221.565,Z 406.749,A -85,B 0,C 180,E1 -21283.309,E2 -21283.309} C_VEL
LIN {X 0,Y 228.461,Z 420.141,A -85,B 0,C 180,E1 -21285.694,E2 -21285.694} C_VEL
LIN {X 0,Y 235.127,Z 435.311,A -85,B 0,C 180,E1 -21287.876,E2 -21287.876} C_VEL
LIN {X 0,Y 236.483,Z 438.606,A -85,B 0,C 180,E1 -21288.304,E2 -21288.304} C_VEL
LIN {X 0,Y 233.424,Z 496.044,A -85,B 0,C 180,E1 -21289.933,E2 -21289.933} C_VEL
LIN {X 0,Y 232.231,Z 513.175,A -85,B 0,C 180,E1 -21290.502,E2 -21290.502} C_VEL
LIN {X 0,Y 230.279,Z 527.795,A -85,B 0,C 180,E1 -21291.273,E2 -21291.273} C_VEL
LIN {X 0,Y 227.839,Z 541.362,A -85,B 0,C 180,E1 -21292.331,E2 -21292.331} C_VEL
LIN {X 0,Y 225.109,Z 553.622,A -85,B 0,C 180,E1 -21293.62,E2 -21293.62} C_VEL
LIN {X 0,Y 221.914,Z 565.694,A -85,B 0,C 180,E1 -21295.249,E2 -21295.249} C_VEL
LIN {X 0,Y 218.618,Z 576.789,A -85,B 0,C 180,E1 -21297.15,E2 -21297.15} C_VEL
LIN {X 0,Y 214.674,Z 587.939,A -85,B 0,C 180,E1 -21299.51,E2 -21299.51} C_VEL
LIN {X 0,Y 210.87,Z 597.942,A -85,B 0,C 180,E1 -21302.189,E2 -21302.189} C_VEL
LIN {X 0,Y 207.49,Z 606.248,A -85,B 0,C 180,E1 -21304.954,E2 -21304.954} C_VEL
LIN {X 0,Y 204.268,Z 614.142,A -85,B 0,C 180,E1 -21308.272,E2 -21308.272} C_VEL
LIN {X 0,Y 201.78,Z 620.574,A -85,B 0,C 180,E1 -21311.734,E2 -21311.734} C_VEL
LIN {X 0,Y 199.413,Z 626.238,A -85,B 0,C 180,E1 -21315.72,E2 -21315.72} C_VEL
LIN {X 0,Y 198.061,Z 630.346,A -85,B 0,C 180,E1 -21319.783,E2 -21319.783} C_VEL
LIN {X 0,Y 197.365,Z 633.022,A -85,B 0,C 180,E1 -21323.87,E2 -21323.87} C_VEL
LIN {X 0,Y 197.199,Z 634.34,A -85,B 0,C 180,E1 -21327.96,E2 -21327.96} C_VEL
LIN {X 0,Y 197.207,Z 634.5,A -85,B 0,C 180,E1 -21330.003,E2 -21330.003} C_VEL
LIN {X 0,Y 197.246,Z 633.824,A -85,B 0,C 180,E1 -21334.089,E2 -21334.089} C_VEL
LIN {X 0,Y 197.755,Z 631.822,A -85,B 0,C 180,E1 -21338.175,E2 -21338.175} C_VEL
LIN {X 0,Y 198.056,Z 631.223,A -85,B 0,C 180,E1 -21339.191,E2 -21339.191} C_VEL
LIN {X 0,Y 199.03,Z 632.614,A -85,B 0,C 180,E1 -21342.234,E2 -21342.234} C_VEL
LIN {X 0,Y 201.271,Z 633.219,A -85,B 0,C 180,E1 -21346.224,E2 -21346.224} C_VEL
LIN {X 0,Y 204.633,Z 632.403,A -85,B 0,C 180,E1 -21350.089,E2 -21350.089} C_VEL
LIN {X 0,Y 208.951,Z 630.224,A -85,B 0,C 180,E1 -21353.807,E2 -21353.807} C_VEL
LIN {X 0,Y 214.459,Z 626.582,A -85,B 0,C 180,E1 -21357.312,E2 -21357.312} C_VEL
LIN {X 0,Y 220.953,Z 621.394,A -85,B 0,C 180,E1 -21360.594,E2 -21360.594} C_VEL
LIN {X 0,Y 226.333,Z 616.469,A -85,B 0,C 180,E1 -21362.918,E2 -21362.918} C_VEL
LIN {X 0,Y 233.326,Z 609.41,A -85,B 0,C 180,E1 -21365.441,E2 -21365.441} C_VEL
LIN {X 0,Y 240.916,Z 600.712,A -85,B 0,C 180,E1 -21367.781,E2 -21367.781} C_VEL
LIN {X 0,Y 249.035,Z 590.151,A -85,B 0,C 180,E1 -21369.945,E2 -21369.945} C_VEL
LIN {X 0,Y 256.121,Z 579.593,A -85,B 0,C 180,E1 -21371.586,E2 -21371.586} C_VEL
LIN {X 0,Y 262.979,Z 567.875,A -85,B 0,C 180,E1 -21372.961,E2 -21372.961} C_VEL
LIN {X 0,Y 269.083,Z 555.718,A -85,B 0,C 180,E1 -21374.061,E2 -21374.061} C_VEL
LIN {X 0,Y 274.669,Z 542.151,A -85,B 0,C 180,E1 -21374.981,E2 -21374.981} C_VEL
LIN {X 0,Y 279.419,Z 527.503,A -85,B 0,C 180,E1 -21375.699,E2 -21375.699} C_VEL
LIN {X 0,Y 279.546,Z 527.051,A -85,B 0,C 180,E1 -21375.715,E2 -21375.715} C_VEL
LIN {X 0,Y 278.293,Z 531.564,A -85,B 0,C 180,E1 -21375.954,E2 -21375.954} C_VEL
LIN {X 0,Y 273.296,Z 546.633,A -85,B 0,C 180,E1 -21376.702,E2 -21376.702} C_VEL
LIN {X 0,Y 268.149,Z 558.93,A -85,B 0,C 180,E1 -21377.535,E2 -21377.535} C_VEL
LIN {X 0,Y 262.309,Z 570.598,A -85,B 0,C 180,E1 -21378.561,E2 -21378.561} C_VEL
LIN {X 0,Y 255.298,Z 582.52,A -85,B 0,C 180,E1 -21379.948,E2 -21379.948} C_VEL
LIN {X 0,Y 248.442,Z 592.669,A -85,B 0,C 180,E1 -21381.513,E2 -21381.513} C_VEL
LIN {X 0,Y 241.404,Z 601.867,A -85,B 0,C 180,E1 -21383.358,E2 -21383.358} C_VEL
LIN {X 0,Y 233.7,Z 610.668,A -85,B 0,C 180,E1 -21385.677,E2 -21385.677} C_VEL
LIN {X 0,Y 226.638,Z 617.777,A -85,B 0,C 180,E1 -21388.186,E2 -21388.186} C_VEL
LIN {X 0,Y 221.087,Z 622.72,A -85,B 0,C 180,E1 -21390.481,E2 -21390.481} C_VEL
LIN {X 0,Y 216.08,Z 626.652,A -85,B 0,C 180,E1 -21392.913,E2 -21392.913} C_VEL
LIN {X 0,Y 212.989,Z 628.792,A -85,B 0,C 180,E1 -21394.599,E2 -21394.599} C_VEL
LIN {X 0,Y 210.179,Z 630.526,A -85,B 0,C 180,E1 -21396.343,E2 -21396.343} C_VEL
LIN {X 0,Y 205.646,Z 632.826,A -85,B 0,C 180,E1 -21400.016,E2 -21400.016} C_VEL
LIN {X 0,Y 202.029,Z 633.733,A -85,B 0,C 180,E1 -21403.842,E2 -21403.842} C_VEL
LIN {X 0,Y 199.487,Z 633.187,A -85,B 0,C 180,E1 -21407.797,E2 -21407.797} C_VEL
LIN {X 0,Y 198.058,Z 631.145,A -85,B 0,C 180,E1 -21411.84,E2 -21411.84} C_VEL
LIN {X 0,Y 197.626,Z 627.596,A -85,B 0,C 180,E1 -21415.922,E2 -21415.922} C_VEL
LIN {X 0,Y 197.707,Z 623.763,A -85,B 0,C 180,E1 -21418.982,E2 -21418.982} C_VEL
LIN {X 0,Y 197.903,Z 618.773,A -85,B 0,C 180,E1 -21422.035,E2 -21422.035} C_VEL
LIN {X 0,Y 198.128,Z 612.407,A -85,B 0,C 180,E1 -21425.088,E2 -21425.088} C_VEL
LIN {X 0,Y 198.512,Z 604.251,A -85,B 0,C 180,E1 -21428.189,E2 -21428.189} C_VEL
LIN {X 0,Y 198.967,Z 596.219,A -85,B 0,C 180,E1 -21430.687,E2 -21430.687} C_VEL
LIN {X 0,Y 199.764,Z 586.353,A -85,B 0,C 180,E1 -21433.22,E2 -21433.22} C_VEL
LIN {X 0,Y 200.646,Z 575.458,A -85,B 0,C 180,E1 -21435.491,E2 -21435.491} C_VEL
LIN {X 0,Y 201.643,Z 563.546,A -85,B 0,C 180,E1 -21437.495,E2 -21437.495} C_VEL
LIN {X 0,Y 202.659,Z 550.374,A -85,B 0,C 180,E1 -21439.236,E2 -21439.236} C_VEL
LIN {X 0,Y 203.571,Z 535.91,A -85,B 0,C 180,E1 -21440.651,E2 -21440.651} C_VEL
LIN {X 0,Y 204.342,Z 520.876,A -85,B 0,C 180,E1 -21441.683,E2 -21441.683} C_VEL
LIN {X 0,Y 207.203,Z 457.729,A -85,B 0,C 180,E1 -21445.531,E2 -21445.531} C_VEL
LIN {X 0,Y 204.922,Z 428.801,A -85,B 0,C 180,E1 -21447.371,E2 -21447.371} C_VEL
LIN {X 0,Y 204.842,Z 419.606,A -85,B 0,C 180,E1 -21447.974,E2 -21447.974} C_VEL
LIN {X 0,Y 206.592,Z 406.022,A -85,B 0,C 180,E1 -21451.397,E2 -21451.397} C_VEL
LIN {X 0,Y 203.585,Z 391.623,A -85,B 0,C 180,E1 -21455.395,E2 -21455.395} C_VEL
LIN {X 0,Y 203.166,Z 389.639,A -85,B 0,C 180,E1 -21456.142,E2 -21456.142} C_VEL
LIN {X 0,Y 203.442,Z 389.537,A -85,B 0,C 180,E1 -21456.685,E2 -21456.685} C_VEL
LIN {X 0,Y 204.493,Z 390.123,A -85,B 0,C 180,E1 -21457.175,E2 -21457.175} C_VEL
LIN {X 0,Y 206.864,Z 389.701,A -85,B 0,C 180,E1 -21458.01,E2 -21458.01} C_VEL
LIN {X 0,Y 207.445,Z 389.317,A -85,B 0,C 180,E1 -21458.194,E2 -21458.194} C_VEL
LIN {X 0,Y 210.809,Z 389.807,A -85,B 0,C 180,E1 -21459.368,E2 -21459.368} C_VEL
LIN {X 0,Y 215.35,Z 396.409,A -85,B 0,C 180,E1 -21461.148,E2 -21461.148} C_VEL
LIN {X 0,Y 221.343,Z 406.628,A -85,B 0,C 180,E1 -21463.37,E2 -21463.37} C_VEL
LIN {X 0,Y 227.22,Z 417.74,A -85,B 0,C 180,E1 -21465.404,E2 -21465.404} C_VEL
LIN {X 0,Y 233.951,Z 432.558,A -85,B 0,C 180,E1 -21467.615,E2 -21467.615} C_VEL
LIN {X 0,Y 236.389,Z 438.575,A -85,B 0,C 180,E1 -21468.393,E2 -21468.393} C_VEL
LIN {X 0,Y 232.441,Z 509.442,A -85,B 0,C 180,E1 -21470.423,E2 -21470.423} C_VEL
LIN {X 0,Y 230.706,Z 524.28,A -85,B 0,C 180,E1 -21471.143,E2 -21471.143} C_VEL
LIN {X 0,Y 228.312,Z 538.194,A -85,B 0,C 180,E1 -21472.138,E2 -21472.138} C_VEL
LIN {X 0,Y 225.589,Z 551.136,A -85,B 0,C 180,E1 -21473.427,E2 -21473.427} C_VEL
LIN {X 0,Y 222.325,Z 563.691,A -85,B 0,C 180,E1 -21475.041,E2 -21475.041} C_VEL
LIN {X 0,Y 218.984,Z 575.144,A -85,B 0,C 180,E1 -21476.933,E2 -21476.933} C_VEL
LIN {X 0,Y 215.426,Z 585.657,A -85,B 0,C 180,E1 -21479.079,E2 -21479.079} C_VEL
LIN {X 0,Y 212.123,Z 594.473,A -85,B 0,C 180,E1 -21481.285,E2 -21481.285} C_VEL
LIN {X 0,Y 208.639,Z 603.361,A -85,B 0,C 180,E1 -21484.027,E2 -21484.027} C_VEL
LIN {X 0,Y 205.11,Z 611.873,A -85,B 0,C 180,E1 -21487.324,E2 -21487.324} C_VEL
LIN {X 0,Y 202.438,Z 618.732,A -85,B 0,C 180,E1 -21490.74,E2 -21490.74} C_VEL
LIN {X 0,Y 200.506,Z 623.466,A -85,B 0,C 180,E1 -21493.713,E2 -21493.713} C_VEL
